	dryingSectionGroup3SteamPressureKp : REAL := 1.0;  // PID Kp for Group 1 steam pressure
	dryingSectionGroup3SteamPressureTn : REAL := 8.0;  // PID Tn for Group 1 steam pressure
	dryingSectionGroup3SteamPressureTv : REAL := 0.0;  // PID Tv for Group 1 steam pressure	

	
	dryingSectionGroup1TorqueKp : REAL := 1.0;  // PID Kp for Group 1 steam pressure
	dryingSectionGroup1TorqueTn : REAL := 8.0;  // PID Tn for Group 1 steam pressure
	dryingSectionGroup1TorqueTv : REAL := 0.0;  // PID Tv for Group 1 steam pressure
	
	dryingSectionGroup2TorqueKp : REAL := 1.0;  // PID Kp for Group 1 steam pressure
	dryingSectionGroup2TorqueTn : REAL := 8.0;  // PID Tn for Group 1 steam pressure
	dryingSectionGroup2TorqueTv : REAL := 0.0;  // PID Tv for Group 1 steam pressure
	
	dryingSectionGroup3TorqueKp : REAL := 1.0;  // PID Kp for Group 1 steam pressure
	dryingSectionGroup3TorqueTn : REAL := 8.0;  // PID Tn for Group 1 steam pressure
	dryingSectionGroup3TorqueTv : REAL := 0.0;  // PID Tv for Group 1 steam pressure
	
	
		
	firstPressDiameter	: REAL := 531.0;
	secondPressDiameter	: REAL := 800.9;	

	formingBoardSuctionRollDiameter		: REAL := 530.0;
	formingBoardTractionRollDiameter	: REAL := 580.0;
    tractionRollToSuctionRollGearRatio  : REAL := 0.915;

	formingBoardSuctionRollMotorRPM		: REAL := 329.3;
	formingBoardTractionRollMotorRPM	: REAL := 360.4;
	formingBoardTorqueDif				: REAL := 1.0;

	
	    //----------------------------------------------------------------------
    // PID GAINS
    //----------------------------------------------------------------------
    formingBoardTorquePIDCtrlKp                   : REAL := 2.0;
    formingBoardTorquePIDCtrlTn                   : REAL := 8.0;
    formingBoardTorquePIDCtrlTv                   : REAL := 0.0;
    formingBoardTorqueLimit                   : REAL := 100.0;
	
	
    pressTorquePIDCtrlKp                   : REAL := 2.0;
    pressTorquePIDCtrlTn                   : REAL := 8.0;
    pressTorquePIDCtrlTv                   : REAL := 0.0;	
    pressTorqueLimit                   	: REAL := 100.0;	
	
    dryingSectionGroup1TorquePIDCtrlKp		: REAL := 2.0;
    dryingSectionGroup1TorquePIDCtrlTn	: REAL := 8.0;
    dryingSectionGroup1TorquePIDCtrlTv	: REAL := 0.0;
    dryingSectionGroup1TorqueLimit	: REAL := 100.0;

		
    dryingSectionGroup2TorquePIDCtrlKp	: REAL := 2.0;
    dryingSectionGroup2TorquePIDCtrlTn	: REAL := 8.0;
    dryingSectionGroup2TorquePIDCtrlTv	: REAL := 0.0;
    dryingSectionGroup2TorqueLimit	: REAL := 100.0;
			
	dryingSectionGroup3TorquePIDCtrlKp	: REAL := 2.0;
    dryingSectionGroup3TorquePIDCtrlTn	: REAL := 8.0;
    dryingSectionGroup3TorquePIDCtrlTv	: REAL := 0.0;
    dryingSectionGroup3TorqueLimit	: REAL := 100.0;
		
	
	

	
	dryingSectionGroup1UpperMasterDiameter	: REAL := 263.878;
	dryingSectionGroup1UpperSlave1Diameter	: REAL := 1200.980;
	dryingSectionGroup1LowerMasterDiameter	: REAL := 263.241;
	dryingSectionGroup1LowerSlave1Diameter	: REAL := 263.241;
	dryingSectionGroup2UpperMasterDiameter	: REAL := 264.196;
	dryingSectionGroup2UpperSlave1Diameter	: REAL := 264.196;
	dryingSectionGroup2LowerMasterDiameter	: REAL := 264.196;
	dryingSectionGroup2LowerSlave1Diameter	: REAL := 264.196;	
	dryingSectionGroup3UpperMasterDiameter	: REAL := 264.196;
	dryingSectionGroup3UpperSlave1Diameter	: REAL := 263.878;
	dryingSectionGroup3LowerMasterDiameter	: REAL := 263.878;
	dryingSectionGroup3LowerSlave1Diameter	: REAL := 263.241;

	
	dryingSectionGroup1UpperAndLowerSpeedCalibration   : REAL := -0.06 ;  // Bias [%] between upper and lower
	dryingSectionGroup2UpperAndLowerSpeedCalibration   : REAL := -0.06 ;  // Bias [%] between upper and lower
	dryingSectionGroup3UpperAndLowerSpeedCalibration   : REAL := -0.06 ;  // Bias [%] between upper and lower
	
	
	dryingSectionGroup1SlaveToMasterRatio	: REAL := 1;
	dryingSectionGroup2SlaveToMasterRatio	: REAL := 1;
	dryingSectionGroup3SlaveToMasterRatio	: REAL := 1;

	dryingSectionGroup1SlaveTorqueDif	: REAL := 1;
	dryingSectionGroup2SlaveTorqueDif	: REAL := 1;
	dryingSectionGroup3SlaveTorqueDif	: REAL := 1;
	

	
	firstPressMotorRPM	: REAL := 374.5;
	secondPressMotorRPM	: REAL := 238.7;	
	
	dryingSectionGroup1UpperMasterMotorRPM	: REAL := 750;
	dryingSectionGroup1UpperSlave1MotorRPM	: REAL := 750;

	dryingSectionGroup1LowerMasterMotorRPM	: REAL := 750;
	dryingSectionGroup1LowerSlave1MotorRPM	: REAL := 750;


	dryingSectionGroup2UpperMasterMotorRPM	: REAL := 750;
	dryingSectionGroup2UpperSlave1MotorRPM	: REAL := 750;

	dryingSectionGroup2LowerMasterMotorRPM	: REAL := 750;
	dryingSectionGroup2LowerSlave1MotorRPM	: REAL := 750;

	
	dryingSectionGroup3UpperMasterMotorRPM	: REAL := 750;
	dryingSectionGroup3UpperSlave1MotorRPM	: REAL := 750;
	
	dryingSectionGroup3LowerMasterMotorRPM	: REAL := 750;
	dryingSectionGroup3LowerSlave1MotorRPM	: REAL := 750;
	
	

	winderDiameter	: REAL := 800.9;
	winderMotorRPM	: REAL := 212.5; //Motor RPM  / Rel. Mecanicia (1700 / 8)
	

	winderRiderRollMovPressure : REAL := 9.0;
	
	
	winderRiderRollStartPressure : REAL := 1.0;
	winderRiderRollAdvTime : TIME := T#2S;

	
			
	END_STRUCT
END_TYPE

// ---- Function Blocks/PaperMachine/DataTypes/PaperMachine_TypeHmiCommands.TcDUT
TYPE PaperMachine_TypeHmiCommands :
STRUCT

    // ─────────────── GENERAL MACHINE COMMANDS ───────────────
    machineReset : BOOL; // General machine reset (Reset geral da máquina)

	
    // ─────────────── FORMING BOARD ───────────────
    formingBoardStart          : BOOL;  // Start forming board (Ligar mesa formadora)
    formingBoardStop           : BOOL;  // Stop forming board (Parar mesa formadora)
    formingBoardFastStop           : BOOL;  // Stop forming board (Parar mesa formadora)

    formingBoardAutoMan           : BOOL;  // Auto mode select (Modo automático)
    formingBoardSetpointMan    : REAL;  // Manual speed/flow setpoint (Setpoint manual)
    formingBoardProductionSpeed: REAL;  // Select production (fast) speed (Selecionar velocidade de produção - rápida)
    formingBoardRollUpCmd      : BOOL;  // Command to raise/roll up forming board (Comando para subir mesa formadora)
    formingBoardRollDownCmd    : BOOL;  // Command to lower/roll down forming board (Comando para descer mesa formadora)

	// Automatic positioning (for auto mode)
	headboxLipsTargetSetpoint_mm       : REAL;          // Desired lips opening [mm]
	headboxLipsAutoAdjustCmd           : BOOL;          // Pulse to start auto adjustment
	// Manual jog commands (for manual mode)
	headboxLipsManualOpenCmd           : BOOL;          // Jog open while pressed
	headboxLipsManualCloseCmd          : BOOL;          // Jog close while pressed		
	
	formingTailCutterNozzleStartCmd   : BOOL; 
	formingTailCutterNozzleStopCmd   : BOOL; 
	
	formingTailCutterNozzleFwCmd   : BOOL; 
	formingTailCutterNozzleRevCmd   : BOOL; 	
	
	
	
	formingWireShowerStartCmd : BOOL; 
	formingWireShowerStopCmd : BOOL; 
	
	
	// ─────────────── PRESS SECTION ───────────────
	// Start/stop and speed control commands for the press section.
	pressSectionStart            : BOOL;  // Start Press Section (Ligar Prensa)
	pressSectionStop             : BOOL;  // Stop Press Section (Parar Prensa)
	pressSectionFastStop             : BOOL;  // Stop Press Section (Parar Prensa)

	pressSectionAutoMan          : BOOL;  // 1 = Auto / 0 = Manual mode (Modo automático/manual)
	pressSectionManualSetpoint   : REAL;  // Manual speed setpoint [m/min] (Setpoint manual)
	pressSectionSpeedInc         : BOOL;  // Increase speed manually (Aumentar velocidade)
	pressSectionSpeedDec         : BOOL;  // Decrease speed manually (Diminuir velocidade)
	pressSectionRecoverSpeedCmd  : BOOL;  // Temporarily recover speed (Recuperar velocidade)
	pressSectionRecoverIncrement : REAL;  // Recovery speed increment [m/min or %] (Incremento de recuperação)

	
	// ─────────────── DRYING SECTION — GROUP 1 ───────────────
	// Start/stop and speed control commands for the drying section (Group 1).
	dryingSectionGroup1Start            : BOOL;  // Start Drying Section Group 1 (Ligar Secagem Grupo 1)
	dryingSectionGroup1Stop             : BOOL;  // Stop Drying Section Group 1 (Parar Secagem Grupo 1)
	dryingSectionGroup1FastStop             : BOOL;  // Stop Drying Section Group 1 (Parar Secagem Grupo 1)

	dryingSectionGroup1AutoMan          : BOOL;  // 1 = Auto / 0 = Manual mode for Group 1 (Modo automático/manual Grupo 1)
	dryingSectionGroup1ManualSetpoint   : REAL;  // Manual speed setpoint [m/min] (Setpoint manual Grupo 1)
	dryingSectionGroup1SpeedInc         : BOOL;  // Increase Group 1 speed manually (Aumentar velocidade Grupo 1)
	dryingSectionGroup1SpeedDec         : BOOL;  // Decrease Group 1 speed manually (Diminuir velocidade Grupo 1)
	dryingSectionGroup1RecoverSpeedCmd  : BOOL;  // Temporarily recover speed (Recuperar velocidade Grupo 1)
	Group1RecoverIncrement : REAL;  // Recovery speed increment [m/min or %] (Incremento de recuperação Grupo 1)
	dryingSectionGroup1SteamPressureAutoMan : BOOL;  // Recovery speed increment [m/min or %] (Incremento de recuperação Grupo 1)
	dryingSectionGroup1SteamPressureAutoSetpoint : REAL;  // Recovery speed increment [m/min or %] (Incremento de recuperação Grupo 1)
	dryingSectionGroup1SteamPressureManualSetpoint : REAL;  // Recovery speed increment [m/min or %] (Incremento de recuperação Grupo 1)
	dryingSectionGroup1PaperBreakSteamPressure1 : REAL;  // Recovery speed increment [m/min or %] (Incremento de recuperação Grupo 1)
	dryingSectionGroup1PaperBreakSteamPressure2 : REAL;  // Recovery speed increment [m/min or %] (Incremento de recuperação Grupo 1)

	
	// ─────────────── DRYING SECTION — GROUP 2 ───────────────
	// Start/stop and speed control commands for the drying section (Group 2).
	dryingSectionGroup2Start            : BOOL;  // Start Drying Section Group 2 (Ligar Secagem Grupo 2)
	dryingSectionGroup2Stop             : BOOL;  // Stop Drying Section Group 2 (Parar Secagem Grupo 2)
	dryingSectionGroup2FastStop             : BOOL;  // Stop Drying Section Group 1 (Parar Secagem Grupo 1)

	dryingSectionGroup2AutoMan          : BOOL;  // 1 = Auto / 0 = Manual mode for Group 2 (Modo automático/manual Grupo 2)

	dryingSectionGroup2ManualSetpoint   : REAL;  // Manual speed setpoint [m/min] (Setpoint manual Grupo 2)
	dryingSectionGroup2SpeedInc         : BOOL;  // Increase Group 2 speed manually (Aumentar velocidade Grupo 2)
	dryingSectionGroup2SpeedDec         : BOOL;  // Decrease Group 2 speed manually (Diminuir velocidade Grupo 2)
	dryingSectionGroup2RecoverSpeedCmd  : BOOL;  // Temporarily recover speed (Recuperar velocidade Grupo 2)
	dryingSectionGroup2RecoverIncrement : REAL;  // Recovery speed increment [m/min or %] (Incremento de recuperação Grupo 2)
	dryingSectionGroup2SteamPressureAutoMan : BOOL;  // Recovery speed increment [m/min or %] (Incremento de recuperação Grupo 1)
	dryingSectionGroup2SteamPressureAutoSetpoint : REAL;  // Recovery speed increment [m/min or %] (Incremento de recuperação Grupo 1)
	dryingSectionGroup2SteamPressureManualSetpoint : REAL;  // Recovery speed increment [m/min or %] (Incremento de recuperação Grupo 1)
	dryingSectionGroup2PaperBreakSteamPressure1 : REAL;  // Recovery speed increment [m/min or %] (Incremento de recuperação Grupo 1)
	dryingSectionGroup2PaperBreakSteamPressure2 : REAL;  // Recovery speed increment [m/min or %] (Incremento de recuperação Grupo 1)
	
	// ─────────────── DRYING SECTION — GROUP 3 ───────────────
	// Start/stop and speed control commands for the drying section (Group 2).
	dryingSectionGroup3Start            : BOOL;  // Start Drying Section Group 2 (Ligar Secagem Grupo 2)
	dryingSectionGroup3Stop             : BOOL;  // Stop Drying Section Group 2 (Parar Secagem Grupo 2)
	dryingSectionGroup3FastStop             : BOOL;  // Stop Drying Section Group 1 (Parar Secagem Grupo 1)

	dryingSectionGroup3AutoMan          : BOOL;  // 1 = Auto / 0 = Manual mode for Group 2 (Modo automático/manual Grupo 2)
	dryingSectionGroup3ManualSetpoint   : REAL;  // Manual speed setpoint [m/min] (Setpoint manual Grupo 2)
	dryingSectionGroup3SpeedInc         : BOOL;  // Increase Group 2 speed manually (Aumentar velocidade Grupo 2)
	dryingSectionGroup3SpeedDec         : BOOL;  // Decrease Group 2 speed manually (Diminuir velocidade Grupo 2)
	dryingSectionGroup3RecoverSpeedCmd  : BOOL;  // Temporarily recover speed (Recuperar velocidade Grupo 2)
	dryingSectionGroup3RecoverIncrement : REAL;  // Recovery speed increment [m/min or %] (Incremento de recuperação Grupo 2)
	dryingSectionGroup3SteamPressureAutoMan : BOOL;  // Recovery speed increment [m/min or %] (Incremento de recuperação Grupo 1)
	dryingSectionGroup3SteamPressureAutoSetpoint : REAL;  // Recovery speed increment [m/min or %] (Incremento de recuperação Grupo 1)
	dryingSectionGroup3SteamPressureManualSetpoint : REAL;  // Recovery speed increment [m/min or %] (Incremento de recuperação Grupo 1)
	dryingSectionGroup3PaperBreakSteamPressure1 : REAL;  // Recovery speed increment [m/min or %] (Incremento de recuperação Grupo 1)
	dryingSectionGroup3PaperBreakSteamPressure2 : REAL;  // Recovery speed increment [m/min or %] (Incremento de recuperação Grupo 1)
	
    // ─────────────── DRYING SECTION - LUBRIFICATION UNIT ───────────────
    dryingSectionLubricationPumpStart      : BOOL;  // EN: Start command for lubrication unit (HMI → FB) / PT: Comando de PARTIDA da unidade de lubrificação (IHM → FB)
    dryingSectionLubricationPumpStop       : BOOL;  // EN: Stop command for lubrication unit (HMI → FB) / PT: Comando de PARADA da unidade de lubrificação (IHM → FB)
    dryingSectionLubricationPumpSelector   : BOOL;  // EN: Pump selector (FALSE = Pump 1, TRUE = Pump 2) / PT: Seletor de bomba (FALSE = Bomba 1, TRUE = Bomba 2)
    dryingSectionLubricationPumpAutoMan    : BOOL;  // EN: Mode selection (FALSE = Manual, TRUE = Automatic) / PT: Seleção de modo (FALSE = Manual, TRUE = Automático)

	// ─────────────── WINDER SECTION ───────────────
	// Start/stop and speed control commands for the winder section.
	winderSectionStart            : BOOL;  // Start Press Section (Ligar Prensa)
	winderSectionStop             : BOOL;  // Stop Press Section (Parar Prensa)
	winderSectionAutoMan          : BOOL;  // 1 = Auto / 0 = Manual mode (Modo automático/manual)
	winderSectionManualSetpoint   : REAL;  // Manual speed setpoint [m/min] (Setpoint manual)
	winderSectionSpeedInc         : BOOL;  // Increase speed manually (Aumentar velocidade)
	winderSectionSpeedDec         : BOOL;  // Decrease speed manually (Diminuir velocidade)
	winderSectionRecoverSpeedCmd  : BOOL;  // Temporarily recover speed (Recuperar velocidade)
	winderSectionRecoverIncrement : REAL;  // Recovery speed increment [m/min or %] (Incremento de recuperação)


	
	
	
  // Pressure fine adjustments for rider roll
    winderPressureOperatorSideIncCmd : BOOL; // EN: Increase operator-side pressure / PT: Aumenta a pressão no lado do operador
    winderPressureOperatorSideDecCmd : BOOL; // EN: Decrease operator-side pressure / PT: Diminui a pressão no lado do operador

    winderPressureDriveSideIncCmd    : BOOL; // EN: Increase drive-side pressure / PT: Aumenta a pressão no lado motriz
    winderPressureDriveSideDecCmd    : BOOL; // EN: Decrease drive-side pressure / PT: Diminui a pressão no lado motriz

	winderRiderRollWorkPositionCmd	: BOOL;
	winderRiderRollReleasePositionCmd	: BOOL;
	winderEnableTorqueControlCmd			: BOOL;

	winderTorqueSetpoint			: REAL;
	
    //==============================================================
    // CORE LOCK (CHUCK LOCKING SYSTEM)
    //==============================================================
    winderCoreLockAutoMan         : BOOL;  // EN: Core lock mode (0=Manual, 1=Auto) / PT: Modo do travamento do mandril (0=Manual, 1=Automático)
    winderCoreLockCmd             : BOOL;  // EN: Lock core chucks / PT: Travar mandril (core chucks)
    winderCoreUnlockCmd           : BOOL;  // EN: Unlock core chucks / PT: Destravar mandril

	//==============================================================
    // CORE LOCK (CHUCK LOCKING SYSTEM)
    //==============================================================
	winderCoreAceleratorEngageCmd : BOOL;
	winderCoreAceleratorDisengageCmd : BOOL;
	
    //==============================================================
    // CORE BRAKE CONTROL
    //==============================================================
    winderCoreBrakeAutoMan        : BOOL;  // EN: Core brake mode (0=Manual, 1=Auto) / PT: Modo de freio do mandril (0=Manual, 1=Automático)
    winderCoreBrakeEnableCmd      : BOOL;  // EN: Enable core brake / PT: Habilita o freio do mandril
    winderCoreBrakeDisableCmd     : BOOL;  // EN: Disable core brake / PT: Desabilita o freio do mandril	
	
	winderCorePositioningArmFwdCmd      : BOOL;  // EN: Command to move arm forward / PT: Comando para avançar o braço posicionador
    winderCorePositioningArmRevCmd      : BOOL;  // EN: Command to move arm backward / PT: Comando para recuar o braço posicionador

    winderCorePositioningArmPosLimitFwd : BOOL;  // EN: Forward limit switch / PT: Fim de curso avançado
    winderCorePositioningArmPosLimitRev : BOOL;  // EN: Reverse limit switch / PT: Fim de curso recuado
	
    // ─────────────── CENTRIFUGAL PRESSURE SCREEN ───────────────
    pressureScreenStart : BOOL;  // Start centrifugal pressure screen (Ligar peneira centrífuga de pressão)
    pressureScreenStop  : BOOL;  // Stop centrifugal pressure screen (Parar peneira centrífuga de pressão)
	

    // ─────────────── COUCH PIT PUMP & MIXER ───────────────
    couchPitPumpStart        : BOOL;  // Start couch pit pump (Ligar bomba do poço da mesa couch)
    couchPitPumpStop         : BOOL;  // Stop couch pit pump (Parar bomba do poço da mesa couch)
    couchPitPumpAutoMan      : BOOL;  // Auto/manual mode select (Seleção automático/manual)
    couchPitPumpSetpointMan  : REAL;  // Manual setpoint (Setpoint manual)
    couchPitPumpSetpointAuto : REAL;  // Auto setpoint (Setpoint automático)
    couchPitMixerStart       : BOOL;  // Start couch pit mixer (Ligar misturador do poço da mesa couch)
    couchPitMixerStop        : BOOL;  // Stop couch pit mixer (Parar misturador do poço da mesa couch)

    // ─────────────── WIRE PIT PUMP ───────────────
    wirePitPumpStart    : BOOL;  // Start wire pit pump (Ligar bomba do poço da mesa plana)
    wirePitPumpStop     : BOOL;  // Stop wire pit pump (Parar bomba do poço da mesa plana)
    wirePitPumpAutoMan  : BOOL;  // Auto/manual mode select (Seleção automático/manual)
    wirePitSetpointMan  : REAL;  // Manual setpoint (Setpoint manual)
    wirePitSetpointManInc  : BOOL;  // Manual setpoint (Setpoint manual)
    wirePitSetpointManDec  : BOOL;  // Manual setpoint (Setpoint manual)	
    wirePitSetpointAuto 	: REAL;  // Auto setpoint (Setpoint automático)
    wirePitSetpointAutoInc  : BOOL;  // Manual setpoint (Setpoint manual)
    wirePitSetpointAutoDec  : BOOL;  // Manual setpoint (Setpoint manual)	

	
	whiteWaterSiloAutoMan           : BOOL;  // Auto/manual mode select (Seleção automático/manual)
	
	// --- Manual setpoint (e.g., level %, flow m3/h, or pressure) ---
	whiteWaterSiloSetpointMan       : REAL;  // Manual setpoint (Setpoint manual)
	whiteWaterSiloSetpointManInc    : BOOL;  // Manual setpoint increase command (Incrementar setpoint manual)
	whiteWaterSiloSetpointManDec    : BOOL;  // Manual setpoint decrease command (Decrementar setpoint manual)
	
	// --- Auto setpoint (from recipe / process / cascade control) ---
	whiteWaterSiloSetpointAuto      : REAL;  // Auto setpoint (Setpoint automático)
	whiteWaterSiloSetpointAutoInc   : BOOL;  // Auto setpoint increase command (Incrementar setpoint automático)
	whiteWaterSiloSetpointAutoDec   : BOOL;  // Auto setpoint decrease command (Decrementar setpoint automático)	
	
	
    // ─────────────── STOCK PUMP ───────────────
    stockPumpStart        : BOOL;  // Start stock pump (Ligar bomba de massa)
    stockPumpStop         : BOOL;  // Stop stock pump (Parar bomba de massa)
    stockPumpAutoMan      : BOOL;  // Auto/manual mode select (Seleção automático/manual)
    stockPumpSetpointMan  : REAL;  // Manual setpoint (Setpoint manual)
    stockPumpSetpointManInc  : BOOL;  // Manual setpoint (Setpoint manual)
    stockPumpSetpointManDec  : BOOL;  // Manual setpoint (Setpoint manual)
	
    stockPumpSetpointAuto : REAL;  // Auto setpoint (Setpoint automático)
    stockPumpSetpointAutoInc : BOOL;  // Auto setpoint (Setpoint automático)
    stockPumpSetpointAutoDec : BOOL;  // Auto setpoint (Setpoint automático)
	

    // ─────────────── MIX PUMP ───────────────
    mixPumpStart      : BOOL;  // Start mixing pump (Ligar bomba de mistura)
    mixPumpStop       : BOOL;  // Stop mixing pump (Parar bomba de mistura)
    mixPumpAutoMan    : BOOL;  // Auto/manual mode select (Seleção automático/manual)
	mixPumpSetpointManInc: BOOL;  // Manual setpoint (Setpoint manual)
	mixPumpSetpointManDec: BOOL;  // Manual setpoint (Setpoint manual)
	mixPumpRatioInc   : BOOL;  // Increase mix ratio (Aumentar proporção de mistura)
    mixPumpRatioDec   : BOOL;  // Decrease mix ratio (Diminuir proporção de mistura)
	mixPumpSetpointMan: REAL;  // Manual setpoint (Setpoint manual)
	mixPumpRatio   	: REAL;  // Increase mix ratio (Aumentar proporção de mistura)

    // ─────────────── VACUUM PUMPS ───────────────
    vacuumSealPumpStart      : BOOL;  // Start vacuum seal pump (Ligar bomba de vedação a vácuo)
    vacuumSealPumpStop       : BOOL;  // Stop vacuum seal pump (Parar bomba de vedação a vácuo)
    vacuumWaterSepPumpStart  : BOOL;  // Start water separator vacuum pump (Ligar bomba de vácuo separadora de água)
    vacuumWaterSepPumpStop   : BOOL;  // Stop water separator vacuum pump (Parar bomba de vácuo separadora de água)
    suctionRollVacuumPumpStart: BOOL; // Start suction roll vacuum pump (Ligar bomba de vácuo do rolo de sucção)
    suctionRollVacuumPumpStop : BOOL; // Stop suction roll vacuum pump (Parar bomba de vácuo do rolo de sucção)
    wireVacuumPumpStart      : BOOL;  // Start wire section vacuum pump (Ligar bomba de vácuo da mesa plana)
    wireVacuumPumpStop       : BOOL;  // Stop wire section vacuum pump (Parar bomba de vácuo da mesa plana)
    pressVacuumPump1Start     : BOOL;  // Start press section vacuum pump (Ligar bomba de vácuo da seção de prensas)
    pressVacuumPump1Stop      : BOOL;  // Stop press section vacuum pump (Parar bomba de vácuo da seção de prensas)
    pressVacuumPump2Start     : BOOL;  // Start press section vacuum pump (Ligar bomba de vácuo da seção de prensas)
    pressVacuumPump2Stop      : BOOL;  // Stop press section vacuum pump (Parar bomba de vácuo da seção de prensas)

    // ─────────────── LOW VACUUM EXHAUST FAN ───────────────
    lowVacuumExhaustFanStart : BOOL;  // Start low vacuum exhaust fan (Ligar exaustor do baixo vácuo)
    lowVacuumExhaustFanStop  : BOOL;  // Stop low vacuum exhaust fan (Parar exaustor do baixo vácuo)

    // ─────────────── WIRE SECTION ───────────────
    wireSectionDisplacementOpSide    : BOOL;  // Displacement sensor - operator side (Sensor de deslocamento - lado operador)
    wireSectionDisplacementDriveSide : BOOL;  // Displacement sensor - drive side (Sensor de deslocamento - lado acionamento)
    wireSectionTensionLimitMax       : REAL;  // Maximum wire tension limit (Limite máximo de tensão da tela formadora)
    wireSectionTensionLimitMin       : REAL;  // Minimum wire tension limit (Limite mínimo de tensão da tela formadora)
    wireSectionStretchExtendCmd      : BOOL;  // Command to stretch wire (Comando para esticar a tela)
    wireSectionStretchReleaseCmd     : BOOL;  // Command to release wire (Comando para aliviar a tela)

END_STRUCT
END_TYPE

// ---- Function Blocks/PaperMachine/DataTypes/PaperMachine_TypeHmiStatus.TcDUT
TYPE PaperMachine_TypeHmiStatus :
STRUCT

	alarmIndication	: BOOL; //Used to tell the hmi that we have an alarm active

    // ─────────────── FORMING LIPS OPENNING CONTROL ───────────────
	headboxLipsPosition_mm       		  : REAL;  // Head box lips position [mm]
	
    // ─────────────── FORMING BOARD ROLLS ───────────────
    formingBoardSuctionRollSpeed    : REAL;  // Suction roll speed (Velocidade do rolo de sucção)
    formingBoardSuctionRollTorque   : REAL;  // Suction roll torque (Torque do rolo de sucção)
    formingBoardSuctionRollState   	: INT;  // Suction roll state 

    formingBoardTractionRollSpeed   : REAL;  // Traction roll speed (Velocidade do rolo tracionador)
    formingBoardTractionRollTorque  : REAL;  // Traction roll torque (Torque do rolo tracionador)
    formingBoardTractionRollState  	: INT;  // Traction roll state 
	
	formingTailCutterNozzleState   : INT; 
	formingWireShowerState : INT; 
	
	// ─────────────── PRESS SECTION DRIVES ───────────────
	firstPressSectionSpeed     : REAL;  // First Press (Master) speed [m/min or rpm] (Velocidade do rolo prensador 1 - mestre)
	firstPressSectionTorque    : REAL;  // First Press (Master) torque [% or Nm] (Torque do rolo prensador 1 - mestre)
	firstPressSectionState     : INT;   // First Press (Master) state code (Estado do rolo prensador 1 - mestre)
	
	secondPressSectionSpeed    : REAL;  // Second Press (Slave) speed [m/min or rpm] (Velocidade do rolo prensador 2 - escravo)
	secondPressSectionTorque   : REAL;  // Second Press (Slave) torque [% or Nm] (Torque do rolo prensador 2 - escravo)
	secondPressSectionState    : INT;   // Second Press (Slave) state code (Estado do rolo prensador 2 - escravo)
	presseGroupSpeedDif				: REAL;	
		
	
	// ─────────────── DRYING SECTION — GROUP 1 ───────────────
	// Speed, torque, and state variables for upper and lower groups of Drying Section Group 1.
	
	// ── UPPER GROUP (GROUP 1) ────────────────────────────────────────────────
	dryingSectionGroup1UpperMasterSpeedMPM   : REAL;  // Group 1 Upper Master speed [m/min or rpm] (Velocidade do motor mestre superior do grupo 1)
	dryingSectionGroup1UpperMasterTorque  : REAL;  // Group 1 Upper Master torque [% or Nm] (Torque do motor mestre superior do grupo 1)
	dryingSectionGroup1UpperMasterState   : INT;   // Group 1 Upper Master state code (Estado do motor mestre superior do grupo 1)
	
	dryingSectionGroup1UpperSlave1SpeedMPM   : REAL;  // Group 1 Upper Slave 1 speed [m/min or rpm] (Velocidade do motor escravo 1 superior do grupo 1)
	dryingSectionGroup1UpperSlave1Torque  : REAL;  // Group 1 Upper Slave 1 torque [% or Nm] (Torque do motor escravo 1 superior do grupo 1)
	dryingSectionGroup1UpperSlave1State   : INT;   // Group 1 Upper Slave 1 state code (Estado do motor escravo 1 superior do grupo 1)
	
	dryingSectionGroup1UpperSlave2SpeedMPM   : REAL;  // Group 1 Upper Slave 2 speed [m/min or rpm] (Velocidade do motor escravo 2 superior do grupo 1)
	dryingSectionGroup1UpperSlave2Torque  : REAL;  // Group 1 Upper Slave 2 torque [% or Nm] (Torque do motor escravo 2 superior do grupo 1)
	dryingSectionGroup1UpperSlave2State   : INT;   // Group 1 Upper Slave 2 state code (Estado do motor escravo 2 superior do grupo 1)
	
	
	// ── LOWER GROUP (GROUP 1) ────────────────────────────────────────────────
	dryingSectionGroup1LowerMasterSpeedMPM   : REAL;  // Group 1 Lower Master speed [m/min or rpm] (Velocidade do motor mestre inferior do grupo 1)
	dryingSectionGroup1LowerMasterTorque  : REAL;  // Group 1 Lower Master torque [% or Nm] (Torque do motor mestre inferior do grupo 1)
	dryingSectionGroup1LowerMasterState   : INT;   // Group 1 Lower Master state code (Estado do motor mestre inferior do grupo 1)
	
	dryingSectionGroup1LowerSlave1SpeedMPM   : REAL;  // Group 1 Lower Slave 1 speed [m/min or rpm] (Velocidade do motor escravo 1 inferior do grupo 1)
	dryingSectionGroup1LowerSlave1Torque  : REAL;  // Group 1 Lower Slave 1 torque [% or Nm] (Torque do motor escravo 1 inferior do grupo 1)
	dryingSectionGroup1LowerSlave1State   : INT;   // Group 1 Lower Slave 1 state code (Estado do motor escravo 1 inferior do grupo 1)
	
	dryingSectionGroup1LowerSlave2SpeedMPM   : REAL;  // Group 1 Lower Slave 2 speed [m/min or rpm] (Velocidade do motor escravo 2 inferior do grupo 1)
	dryingSectionGroup1LowerSlave2Torque  : REAL;  // Group 1 Lower Slave 2 torque [% or Nm] (Torque do motor escravo 2 inferior do grupo 1)
	dryingSectionGroup1LowerSlave2State   : INT;   // Group 1 Lower Slave 2 state code (Estado do motor escravo 2 inferior do grupo 1)
	
	dryingSectionGroup1SteamPressure   : REAL;   // Drying group 1 - Steam pressure display
	dryingSectionGroup1SpeedDif				: REAL;	

	dryingSectionGroup1PaperPresence				: BOOL;	
	
	
	// ─────────────── DRYING SECTION — GROUP 2 ───────────────
	// Speed, torque, and state variables for upper and lower groups of Drying Section Group 2.
	
	// ── UPPER GROUP (GROUP 2) ────────────────────────────────────────────────
	dryingSectionGroup2UpperMasterSpeedMPM   : REAL;  // Group 2 Upper Master speed [m/min or rpm] (Velocidade do motor mestre superior do grupo 2)
	dryingSectionGroup2UpperMasterTorque  : REAL;  // Group 2 Upper Master torque [% or Nm] (Torque do motor mestre superior do grupo 2)
	dryingSectionGroup2UpperMasterState   : INT;   // Group 2 Upper Master state code (Estado do motor mestre superior do grupo 2)
	
	dryingSectionGroup2UpperSlave1SpeedMPM   : REAL;  // Group 2 Upper Slave 1 speed [m/min or rpm] (Velocidade do motor escravo 1 superior do grupo 2)
	dryingSectionGroup2UpperSlave1Torque  : REAL;  // Group 2 Upper Slave 1 torque [% or Nm] (Torque do motor escravo 1 superior do grupo 2)
	dryingSectionGroup2UpperSlave1State   : INT;   // Group 2 Upper Slave 1 state code (Estado do motor escravo 1 superior do grupo 2)
	
	dryingSectionGroup2UpperSlave2Speed   : REAL;  // Group 2 Upper Slave 2 speed [m/min or rpm] (Velocidade do motor escravo 2 superior do grupo 2)
	dryingSectionGroup2UpperSlave2Torque  : REAL;  // Group 2 Upper Slave 2 torque [% or Nm] (Torque do motor escravo 2 superior do grupo 2)
	dryingSectionGroup2UpperSlave2State   : INT;   // Group 2 Upper Slave 2 state code (Estado do motor escravo 2 superior do grupo 2)
	
	
	// ── LOWER GROUP (GROUP 2) ────────────────────────────────────────────────
	dryingSectionGroup2LowerMasterSpeedMPM   : REAL;  // Group 2 Lower Master speed [m/min or rpm] (Velocidade do motor mestre inferior do grupo 2)
	dryingSectionGroup2LowerMasterTorque  : REAL;  // Group 2 Lower Master torque [% or Nm] (Torque do motor mestre inferior do grupo 2)
	dryingSectionGroup2LowerMasterState   : INT;   // Group 2 Lower Master state code (Estado do motor mestre inferior do grupo 2)
	
	dryingSectionGroup2LowerSlave1SpeedMPM   : REAL;  // Group 2 Lower Slave 1 speed [m/min or rpm] (Velocidade do motor escravo 1 inferior do grupo 2)
	dryingSectionGroup2LowerSlave1Torque  : REAL;  // Group 2 Lower Slave 1 torque [% or Nm] (Torque do motor escravo 1 inferior do grupo 2)
	dryingSectionGroup2LowerSlave1State   : INT;   // Group 2 Lower Slave 1 state code (Estado do motor escravo 1 inferior do grupo 2)
	
	dryingSectionGroup2LowerSlave2SpeedMPM   : REAL;  // Group 2 Lower Slave 2 speed [m/min or rpm] (Velocidade do motor escravo 2 inferior do grupo 2)
	dryingSectionGroup2LowerSlave2Torque  : REAL;  // Group 2 Lower Slave 2 torque [% or Nm] (Torque do motor escravo 2 inferior do grupo 2)
	dryingSectionGroup2LowerSlave2State   : INT;   // Group 2 Lower Slave 2 state code (Estado do motor escravo 2 inferior do grupo 2)
	
	dryingSectionGroup2SteamPressure   : REAL;   // Drying group 1 - Steam pressure display
	dryingSectionGroup2SpeedDif				: REAL;	
		
	dryingSectionGroup2PaperPresence				: BOOL;	
	
	// ─────────────── DRYING SECTION — GROUP 3 ───────────────
	// Speed, torque, and state variables for upper and lower groups of Drying Section Group 2.
	
	// ── UPPER GROUP (GROUP 3) ────────────────────────────────────────────────
	dryingSectionGroup3UpperMasterSpeedMPM   : REAL;  // Group 2 Upper Master speed [m/min or rpm] (Velocidade do motor mestre superior do grupo 2)
	dryingSectionGroup3UpperMasterTorque  : REAL;  // Group 2 Upper Master torque [% or Nm] (Torque do motor mestre superior do grupo 2)
	dryingSectionGroup3UpperMasterState   : INT;   // Group 2 Upper Master state code (Estado do motor mestre superior do grupo 2)
	
	dryingSectionGroup3UpperSlave1SpeedMPM   : REAL;  // Group 2 Upper Slave 1 speed [m/min or rpm] (Velocidade do motor escravo 1 superior do grupo 2)
	dryingSectionGroup3UpperSlave1Torque  : REAL;  // Group 2 Upper Slave 1 torque [% or Nm] (Torque do motor escravo 1 superior do grupo 2)
	dryingSectionGroup3UpperSlave1State   : INT;   // Group 2 Upper Slave 1 state code (Estado do motor escravo 1 superior do grupo 2)
	
	dryingSectionGroup3UpperSlave2SpeedMPM   : REAL;  // Group 2 Upper Slave 2 speed [m/min or rpm] (Velocidade do motor escravo 2 superior do grupo 2)
	dryingSectionGroup3UpperSlave2Torque  : REAL;  // Group 2 Upper Slave 2 torque [% or Nm] (Torque do motor escravo 2 superior do grupo 2)
	dryingSectionGroup3UpperSlave2State   : INT;   // Group 2 Upper Slave 2 state code (Estado do motor escravo 2 superior do grupo 2)
	
	
	// ── LOWER GROUP (GROUP 3) ────────────────────────────────────────────────
	dryingSectionGroup3LowerMasterSpeedMPM   : REAL;  // Group 2 Lower Master speed [m/min or rpm] (Velocidade do motor mestre inferior do grupo 2)
	dryingSectionGroup3LowerMasterTorque  : REAL;  // Group 2 Lower Master torque [% or Nm] (Torque do motor mestre inferior do grupo 2)
	dryingSectionGroup3LowerMasterState   : INT;   // Group 2 Lower Master state code (Estado do motor mestre inferior do grupo 2)
	
	dryingSectionGroup3LowerSlave1SpeedMPM   : REAL;  // Group 2 Lower Slave 1 speed [m/min or rpm] (Velocidade do motor escravo 1 inferior do grupo 2)
	dryingSectionGroup3LowerSlave1Torque  : REAL;  // Group 2 Lower Slave 1 torque [% or Nm] (Torque do motor escravo 1 inferior do grupo 2)
	dryingSectionGroup3LowerSlave1State   : INT;   // Group 2 Lower Slave 1 state code (Estado do motor escravo 1 inferior do grupo 2)
	
	dryingSectionGroup3LowerSlave2SpeedMPM   : REAL;  // Group 2 Lower Slave 2 speed [m/min or rpm] (Velocidade do motor escravo 2 inferior do grupo 2)
	dryingSectionGroup3LowerSlave2Torque  : REAL;  // Group 2 Lower Slave 2 torque [% or Nm] (Torque do motor escravo 2 inferior do grupo 2)
	dryingSectionGroup3LowerSlave2State   : INT;   // Group 2 Lower Slave 2 state code (Estado do motor escravo 2 inferior do grupo 2)

	dryingSectionGroup3SteamPressure   : REAL;   // Drying group 1 - Steam pressure display
	dryingSectionGroup3SpeedDif				: REAL;	
	dryingSectionGroup3PaperPresence				: BOOL;	
	
	
	winderPaperPresence				: BOOL;	

			
    // ─────────────── LUBRIFICATION UNIT ───────────────
    dryingSectionLubricationPump1State             : INT;   // EN: Pump 1 state (0=Stopped,1=Running,3=Fault) / PT: Estado da bomba 1 (0=Parada,1=Rodando,3=Falha)
    dryingSectionLubricationPump2State             : INT;   // EN: Pump 2 state (0=Stopped,1=Running,3=Fault) / PT: Estado da bomba 2 (0=Parada,1=Rodando,3=Falha)
    dryingSectionLubricationTankTemperature        : REAL;  // EN: Oil tank temperature [°C] / PT: Temperatura do tanque de óleo [°C]
    dryingSectionLubricationCircuitTemperature        : REAL;  // EN: Oil tank temperature [°C] / PT: Temperatura do tanque de óleo [°C]	
 
   // ─────────────── CENTRIFUGAL PRESSURE SCREEN ───────────────
    pressureScreenState             : INT;   // Centrifugal pressure screen state (Estado da peneira centrífuga de pressão)


    // ─────────────── COUCH PIT PUMP & MIXER ───────────────
    couchPitPumpState               : INT;   // Couch pit pump state (Estado da bomba do poço da mesa couch)
    couchPitPumpSpeed               : REAL;  // Couch pit pump speed (Velocidade da bomba do poço da mesa couch)
    couchPitPumpTorque              : REAL;  // Couch pit pump torque (Torque da bomba do poço da mesa couch)

    couchPitMixerState              : INT;   // Couch pit mixer state (Estado do agitador do poço da mesa couch)
    couchPitLevel             : REAL;  // Couch pit pump torque (Torque da bomba do poço da mesa couch)


    // ─────────────── WIRE PIT PUMP ───────────────
    wirePitPumpState                : INT;   // Wire pit pump state (Estado da bomba do poço da mesa plana)
    wirePitPumpSpeed                : REAL;  // Wire pit pump speed (Velocidade da bomba do poço da mesa plana)
    wirePitPumpTorque               : REAL;  // Wire pit pump torque (Torque da bomba do poço da mesa plana)
   	wirePitLevel             		: REAL;  // Couch pit pump torque (Torque da bomba do poço da mesa couch)

	
	// --- Manual setpoint (e.g., level %, flow m3/h, or pressure) ---
	whiteWaterSiloLevel       : REAL;  // Manual setpoint (Setpoint manual)
	whiteWaterSiloCtrlOutput       : REAL;  // Manual setpoint (Setpoint manual)

	

    // ─────────────── STOCK PUMP ───────────────
    stockPumpState                  : INT;   // Stock pump state (Estado da bomba de massa)
    stockPumpSpeed               	: REAL;  // Stock pump speed (Velocidade da bomba de massa)
    stockPumpTorque              	: REAL;  // Stock pump torque (Torque da bomba de massa)


    // ─────────────── MIXING PUMP ───────────────
    mixPumpState                    : INT;   // Mixing pump state (Estado da bomba de mistura)
    mixPumpSpeed                    : REAL;  // Mixing pump speed (Velocidade da bomba de mistura)
    mixPumpTorque                   : REAL;  // Mixing pump torque (Torque da bomba de mistura)
 	mixPumpSetpointMan				: REAL;  // Manual setpoint (Setpoint manual)

    // ─────────────── HEAD BOX ───────────────
	
    headBoxMMH2O                    : REAL;  // Pressure in mmH₂O (Pressão em mmH₂O)
    headBoxMMH2OCalc                : REAL;  // Calculated pressure in mmH₂O (Pressão calculada em mmH₂O)
    headBoxJetSpeedMPS                : REAL;  // Calculated pressure in mmH₂O (Pressão calculada em mmH₂O)
	
    mixPumpRatio                    : REAL;  // Mixing ratio (Relação de jato tela)
	
	

    // ─────────────── VACUUM PUMPS ───────────────
    vacuumSealPumpState             : INT;   // Vacuum seal pump state (Estado da bomba de vedação a vácuo)
    vacuumWaterSepPumpState         : INT;   // Water separator vacuum pump state (Estado da bomba de vácuo separadora de água)
    suctionRollVacuumPumpState      : INT;   // Suction roll vacuum pump state (Estado da bomba de vácuo do rolo de sucção)
    wireVacuumPumpState             : INT;   // Wire section vacuum pump state (Estado da bomba de vácuo da mesa plana)


	pressFeltVaccum1State			: INT;
	pressFeltVaccum2State			: INT;
	
	
    // ─────────────── LOW VACUUM EXHAUST FAN ───────────────
    lowVacuumExhaustFanState        : INT;   // Low vacuum exhaust fan state (Estado do exaustor de baixo vácuo)
	
	
	
	winderPressureSetpointOperatorSide : REAL; // EN: Controller output (operator side) / PT: Saída do controlador (lado operador)
    winderPressureSetpointDriveSide    : REAL; // EN: Controller output (drive side) / PT: Saída do controlador (lado motriz)
	winderSpeedMPM   : REAL;  // Group 2 Upper Slave 2 speed [m/min or rpm] (Velocidade do motor escravo 2 superior do grupo 2)
	winderTorque  : REAL;  // Group 2 Upper Slave 2 torque [% or Nm] (Torque do motor escravo 2 superior do grupo 2)
	winderState   : INT;   // Group 2 Upper Slave 2 state code (Estado do motor escravo 2 superior do grupo 2)
	winderSpeedDif				: REAL;	
		

	
	
END_STRUCT
END_TYPE

// ---- Function Blocks/PaperMachine/DataTypes/PaperMachine_TypeHmiAlarms.TcDUT
TYPE PaperMachine_TypeHmiAlarms :
STRUCT

	alarmIndication	: BOOL; //Used to tell the hmi that we have an alarm active

	
	formingBoardSafetyAlarm			: BOOL;
	pressSectionSafetyAlarm			: BOOL;
	dryingSectionSafetyAlarm		: BOOL;
	winderSectionSafetyAlarm		: BOOL;
	
    // ─────────────── FORMING BOARD ROLLS ───────────────
    formingBoardSuctionRollFaultAlarm         : BOOL;  // Suction roll fault / trip
    formingBoardSuctionRollCoolingFaultAlarm  : BOOL;  // Suction roll forced cooling fault
    formingBoardTractionRollFaultAlarm        : BOOL;  // Traction roll fault / trip
    formingBoardTractionRollCoolingFaultAlarm : BOOL;  // Traction roll forced cooling fault

    formingBoardRollDriveFaultAlarm           : BOOL;  // Roll up/down motor fault
    formingBoardStretchDriveFaultAlarm        : BOOL;  // Stretch motor fault
	formingBoardSpeedDifAlarm	: BOOL;

    // ── WIRE EDGE / RUNNING SAFETY SENSORS ─────────────────────────────────────
    formingBoardWireOverrunOperatorSideAlarm  : BOOL;  // Wire overrun detected on operator side (sensor active)
    formingBoardWireOverrunDriveSideAlarm     : BOOL;  // Wire overrun detected on drive side (sensor active)

    // ─────────────── PRESS SECTION DRIVES ───────────────
    pressSectionFirstPressFaultAlarm          : BOOL;  // First press (master) fault / trip
    pressSectionFirstPressCoolingFaultAlarm   : BOOL;  // First press forced cooling fault
    pressSectionSecondPressFaultAlarm         : BOOL;  // Second press (slave) fault / trip
    pressSectionSecondPressCoolingFaultAlarm  : BOOL;  // Second press forced cooling fault

    // ─────────────── PRESS SECTION — AUXILIARY MOTORS ───────────────
    pressSectionUpperFeltStretcherFaultAlarm  : BOOL;  // Upper felt stretcher motor fault / trip
    pressSectionLowerFeltStretcherFaultAlarm  : BOOL;  // Lower felt stretcher motor fault / trip
    pressSectionUpperInfeedRollFaultAlarm     : BOOL;  // Upper infeed roll motor fault / trip
    pressSectionLowerInfeedRollFaultAlarm     : BOOL;  // Lower infeed roll motor fault / trip

    // ── FELT EDGE / RUNNING SAFETY SENSORS ─────────────────────────────────────
    pressSectionUpperFelt1OverrunOperatorSideAlarm : BOOL;  // Felt 1 overrun detected on operator side (sensor active)
    pressSectionUpperFelt1OverrunDriveSideAlarm    : BOOL;  // Felt 1 overrun detected on drive side (sensor active)
    pressSectionUpperFelt2OverrunOperatorSideAlarm : BOOL;  // Felt 2 overrun detected on operator side (sensor active)
    pressSectionUpperFelt2OverrunDriveSideAlarm    : BOOL;  // Felt 2 overrun detected on drive side (sensor active)
    pressSectionLowerFeltOverrunOperatorSideAlarm  : BOOL;  // Felt 3 overrun detected on operator side (sensor active)
    pressSectionLowerFeltOverrunDriveSideAlarm     : BOOL;  // Felt 3 overrun detected on drive side (sensor active)

    // ─────────────── PRESS SECTION — GROUP FAULT ───────────────
    pressSectionGroupFaultAlarm               : BOOL;  // Global press section group fault / interlock active

    // ─────────────── DRYING SECTION — GROUP 1 ───────────────
    dryingSectionGroup1UpperMasterFaultAlarm         : BOOL;  // G1 Upper Master fault / trip
    dryingSectionGroup1UpperMasterCoolingFaultAlarm  : BOOL;  // G1 Upper Master forced cooling fault
    dryingSectionGroup1UpperSlave1FaultAlarm         : BOOL;  // G1 Upper Slave1 fault / trip
    dryingSectionGroup1UpperSlave1CoolingFaultAlarm  : BOOL;  // G1 Upper Slave1 forced cooling fault
    dryingSectionGroup1UpperSlave2FaultAlarm         : BOOL;  // G1 Upper Slave2 fault / trip
    dryingSectionGroup1UpperSlave2CoolingFaultAlarm  : BOOL;  // G1 Upper Slave2 forced cooling fault

    dryingSectionGroup1LowerMasterFaultAlarm         : BOOL;  // G1 Lower Master fault / trip
    dryingSectionGroup1LowerMasterCoolingFaultAlarm  : BOOL;  // G1 Lower Master forced cooling fault
    dryingSectionGroup1LowerSlave1FaultAlarm         : BOOL;  // G1 Lower Slave1 fault / trip
    dryingSectionGroup1LowerSlave1CoolingFaultAlarm  : BOOL;  // G1 Lower Slave1 forced cooling fault
    dryingSectionGroup1LowerSlave2FaultAlarm         : BOOL;  // G1 Lower Slave2 fault / trip
    dryingSectionGroup1LowerSlave2CoolingFaultAlarm  : BOOL;  // G1 Lower Slave2 forced cooling fault

    // ── FABRIC OVERRUN PROTECTION — GROUP 1 ───────────────────────────────────
    upperDryingSectionGroup1FabricOverrunOperatorSideAlarm : BOOL;  // Fabric overrun detected on operator side (sensor active)
    upperDryingSectionGroup1FabricOverrunDriveSideAlarm    : BOOL;  // Fabric overrun detected on drive side (sensor active)
    lowerDryingSectionGroup1FabricOverrunOperatorSideAlarm : BOOL;  // Fabric overrun detected on operator side (sensor active)
    lowerDryingSectionGroup1FabricOverrunDriveSideAlarm    : BOOL;  // Fabric overrun detected on drive side (sensor active)

    // ───────── DRYING SECTION — FABRIC STRETCHER — GROUP 1 ─────────
    upperDryingSectionGroup1FabricStretcherMotorFaultAlarm : BOOL;  // Upper fabric stretcher motor fault (G1)
    lowerDryingSectionGroup1FabricStretcherMotorFaultAlarm : BOOL;  // Lower fabric stretcher motor fault (G1)

    // ───────── DRYING SECTION — AUXILIARIES — GROUP 1 ─────────
    dryingSectionGroup1PickUpRollPosFaultAlarm       : BOOL;  // EN: G1 pick-up roll positioner fault / PT: Falha do posicionador do rolo pick-up G1
    dryingSectionGroup1BabyDryerScraperOscFaultAlarm : BOOL;  // EN: G1 babydryer scraper oscillator fault / PT: Falha do oscilador da raspa do babydryer G1
    dryingSectionGroup1UpperScraperOscFaultAlarm     : BOOL;  // EN: G1 upper group scraper oscillator fault / PT: Falha do oscilador da raspa do grupo superior G1
    dryingSectionGroup1LowerScraperOscFaultAlarm     : BOOL;  // EN: G1 lower group scraper oscillator fault / PT: Falha do oscilador da raspa do grupo inferior G1
	dryingSectionGroup1PaperBreakAlarm : BOOL;

    // ─────────────── DRYING SECTION — GROUP 2 ───────────────
    dryingSectionGroup2UpperMasterFaultAlarm         : BOOL;  // G2 Upper Master fault / trip
    dryingSectionGroup2UpperMasterCoolingFaultAlarm  : BOOL;  // G2 Upper Master forced cooling fault
    dryingSectionGroup2UpperSlave1FaultAlarm         : BOOL;  // G2 Upper Slave1 fault / trip
    dryingSectionGroup2UpperSlave1CoolingFaultAlarm  : BOOL;  // G2 Upper Slave1 forced cooling fault
    dryingSectionGroup2UpperSlave2FaultAlarm         : BOOL;  // G2 Upper Slave2 fault / trip
    dryingSectionGroup2UpperSlave2CoolingFaultAlarm  : BOOL;  // G2 Upper Slave2 forced cooling fault

    dryingSectionGroup2LowerMasterFaultAlarm         : BOOL;  // G2 Lower Master fault / trip
    dryingSectionGroup2LowerMasterCoolingFaultAlarm  : BOOL;  // G2 Lower Master forced cooling fault
    dryingSectionGroup2LowerSlave1FaultAlarm         : BOOL;  // G2 Lower Slave1 fault / trip
    dryingSectionGroup2LowerSlave1CoolingFaultAlarm  : BOOL;  // G2 Lower Slave1 forced cooling fault
    dryingSectionGroup2LowerSlave2FaultAlarm         : BOOL;  // G2 Lower Slave2 fault / trip
    dryingSectionGroup2LowerSlave2CoolingFaultAlarm  : BOOL;  // G2 Lower Slave2 forced cooling fault

    // ── FABRIC OVERRUN PROTECTION — GROUP 2 ───────────────────────────────────
    upperDryingSectionGroup2FabricOverrunOperatorSideAlarm : BOOL;  // Fabric overrun detected on operator side (sensor active)
    upperDryingSectionGroup2FabricOverrunDriveSideAlarm    : BOOL;  // Fabric overrun detected on drive side (sensor active)
    lowerDryingSectionGroup2FabricOverrunOperatorSideAlarm : BOOL;  // Fabric overrun detected on operator side (sensor active)
    lowerDryingSectionGroup2FabricOverrunDriveSideAlarm    : BOOL;  // Fabric overrun detected on drive side (sensor active)

    // ───────── DRYING SECTION — FABRIC STRETCHER — GROUP 2 ─────────
    upperDryingSectionGroup2FabricStretcherMotorFaultAlarm : BOOL;  // Upper fabric stretcher motor fault (G2)
    lowerDryingSectionGroup2FabricStretcherMotorFaultAlarm : BOOL;  // Lower fabric stretcher motor fault (G2)

    // ───────── DRYING SECTION — AUXILIARIES — GROUP 2 ─────────
    dryingSectionGroup2PickUpRollPosFaultAlarm       : BOOL;  // EN: G2 pick-up roll positioner fault / PT: Falha do posicionador do rolo pick-up G2
    dryingSectionGroup2BabyDryerScraperOscFaultAlarm : BOOL;  // EN: G2 babydryer scraper oscillator fault / PT: Falha do oscilador da raspa do babydryer G2
    dryingSectionGroup2UpperScraperOscFaultAlarm     : BOOL;  // EN: G2 upper group scraper oscillator fault / PT: Falha do oscilador da raspa do grupo superior G2
    dryingSectionGroup2LowerScraperOscFaultAlarm     : BOOL;  // EN: G2 lower group scraper oscillator fault / PT: Falha do oscilador da raspa do grupo inferior G2
	dryingSectionGroup2PaperBreakAlarm : BOOL;

    // ─────────────── DRYING SECTION — GROUP 3 ───────────────
    dryingSectionGroup3UpperMasterFaultAlarm         : BOOL;  // G3 Upper Master fault / trip
    dryingSectionGroup3UpperMasterCoolingFaultAlarm  : BOOL;  // G3 Upper Master forced cooling fault
    dryingSectionGroup3UpperSlave1FaultAlarm         : BOOL;  // G3 Upper Slave1 fault / trip
    dryingSectionGroup3UpperSlave1CoolingFaultAlarm  : BOOL;  // G3 Upper Slave1 forced cooling fault
    dryingSectionGroup3UpperSlave2FaultAlarm         : BOOL;  // G3 Upper Slave2 fault / trip
    dryingSectionGroup3UpperSlave2CoolingFaultAlarm  : BOOL;  // G3 Upper Slave2 forced cooling fault

    dryingSectionGroup3LowerMasterFaultAlarm         : BOOL;  // G3 Lower Master fault / trip
    dryingSectionGroup3LowerMasterCoolingFaultAlarm  : BOOL;  // G3 Lower Master forced cooling fault
    dryingSectionGroup3LowerSlave1FaultAlarm         : BOOL;  // G3 Lower Slave1 fault / trip
    dryingSectionGroup3LowerSlave1CoolingFaultAlarm  : BOOL;  // G3 Lower Slave1 forced cooling fault
    dryingSectionGroup3LowerSlave2FaultAlarm         : BOOL;  // G3 Lower Slave2 fault / trip
    dryingSectionGroup3LowerSlave2CoolingFaultAlarm  : BOOL;  // G3 Lower Slave2 forced cooling fault

    // ── FABRIC OVERRUN PROTECTION — GROUP 3 ───────────────────────────────────
    upperDryingSectionGroup3FabricOverrunOperatorSideAlarm : BOOL;  // Fabric overrun detected on operator side (sensor active)
    upperDryingSectionGroup3FabricOverrunDriveSideAlarm    : BOOL;  // Fabric overrun detected on drive side (sensor active)
    lowerDryingSectionGroup3FabricOverrunOperatorSideAlarm : BOOL;  // Fabric overrun detected on operator side (sensor active)
    lowerDryingSectionGroup3FabricOverrunDriveSideAlarm    : BOOL;  // Fabric overrun detected on drive side (sensor active)

    // ───────── DRYING SECTION — FABRIC STRETCHER — GROUP 3 ─────────
    upperDryingSectionGroup3FabricStretcherMotorFaultAlarm : BOOL;  // Upper fabric stretcher motor fault (G3)
    lowerDryingSectionGroup3FabricStretcherMotorFaultAlarm : BOOL;  // Lower fabric stretcher motor fault (G3)

    // ───────── DRYING SECTION — AUXILIARIES — GROUP 3 ─────────
    dryingSectionGroup3PickUpRollPosFaultAlarm       : BOOL;  // EN: G3 pick-up roll positioner fault / PT: Falha do posicionador do rolo pick-up G3
    dryingSectionGroup3BabyDryerScraperOscFaultAlarm : BOOL;  // EN: G3 babydryer scraper oscillator fault / PT: Falha do oscilador da raspa do babydryer G3
    dryingSectionGroup3UpperScraperOscFaultAlarm     : BOOL;  // EN: G3 upper group scraper oscillator fault / PT: Falha do oscilador da raspa do grupo superior G3
    dryingSectionGroup3LowerScraperOscFaultAlarm     : BOOL;  // EN: G3 lower group scraper oscillator fault / PT: Falha do oscilador da raspa do grupo inferior G3
	dryingSectionGroup3PaperBreakAlarm : BOOL;
    // ─────────────── CENTRIFUGAL PRESSURE SCREEN ───────────────
    cpsUnitFaultAlarm                        : BOOL;  // Screen unit fault / trip

    // ─────────────── COUCH PIT PUMP & MIXER ───────────────
    couchPitPumpFaultAlarm                   : BOOL;  // Couch pit pump fault / trip

    // ─────────────── WIRE PIT PUMP ───────────────
    wirePitPumpFaultAlarm                    : BOOL;  // Wire pit pump fault / trip

    // ─────────────── STOCK PUMP ───────────────
    stockPumpFaultAlarm                      : BOOL;  // Stock pump fault / trip

    // ─────────────── MIXING PUMP ───────────────
    mixingPumpFaultAlarm                     : BOOL;  // Mixing pump fault / trip

    // ─────────────── VACUUM PUMPS ───────────────
    vacuumPump1FaultAlarm                    : BOOL;  // Vacuum pump 1 fault / trip
    vacuumPump2FaultAlarm                    : BOOL;  // Vacuum pump 2 fault / trip

    // ─────────────── LOW VACUUM EXHAUST FAN ───────────────
    lowVacuumFanFaultAlarm                   : BOOL;  // Low vacuum exhaust fan fault / trip

    // ─────────────── LUBRIFICATION PUMPS ───────────────
    lubricationPump1FaultAlarm              : BOOL;  // Lubrication pump 1 fault / trip
    lubricationPump2FaultAlarm              : BOOL;  // Lubrication pump 2 fault / trip
    lubricationMinPressureFaultAlarm        : BOOL;  // Minimum pressure not reached / trip
    lubricationMaxPressureFaultAlarm        : BOOL;  // Overpressure in lubrication circuit / trip
	lubricationTankHighTemperatureAlarm 	: BOOL;
	lubricationCircuitHighTemperatureAlarm 	: BOOL;

END_STRUCT
END_TYPE

// ---- Function Blocks/Rewinder/DataTypes/Rewinder_TypePressRoll.TcDUT
TYPE Rewinder_TypePressRoll :
	STRUCT
			
		rollDiameter	: REAL := 0.00;			//Forming board manual speed (Slow speed)
		pressureSetpoint	: REAL := 0.00;			//Forming board manual speed (Slow speed)
				
	END_STRUCT
END_TYPE

// ---- Function Blocks/Rewinder/DataTypes/Rewinder_TypeBrakeControl.TcDUT
TYPE Rewinder_TypeBrakeControl :
	STRUCT
		
	
		rollDiameter		: REAL;			//Forming board manual speed (Slow speed)
		pressureSetpoint	: REAL;			//Forming board manual speed (Slow speed)
		tensionSetpoint		: REAL;
			
	END_STRUCT
END_TYPE

// ---- POUs/MAIN.TcPOU
PROGRAM MAIN
VAR
	instFB_DryingSectionLubrificationControl_V1 : FB_DryingSectionLubrificationControl_V1;
	instFB_SavePersistentData	: FB_SavePersistentData;
	instFB_SpeedDroopControlMst : FB_SpeedDroopControl_1;
	instFB_SpeedDroopControlSlv : FB_FormingBoardDriveControl;
	instFB_DryingSectionDriveControl_GR1 : FB_DryingSectionDriveControl_V1;
	instFB_DryingSectionDriveControl_GR2 : FB_DryingSectionDriveControl_V1;
	
	instFFB_PressSectionDriveControl_V1 : FB_PressSectionDriveControl_V2;
	
	                 

	FB_SoftstarterWithBypass_0: FB_SoftstarterWithBypass;
	FB_PressureControl_0: FB_PressureControl;
	FB_MixPumpControl_0: FB_MixPumpControl;
	FB_HeadboxLipsPWMControl_0: FB_HeadboxLipsPWMControl;
	instPWM: CTRL_PWM;
	instFB_MixPumpControl: FB_MixPumpControl;
	instFB_FormingBoardRollUpDown: FB_FormingBoardRollUpDown;
	instFB_HeadboxLipsPWMControl: FB_HeadboxLipsPWMControl;
	instFB_FormingBoarWireStrech: FB_FormingBoardRollUpDown;
	instFB_FormingBoardWireStretchControl: FB_FormingBoardWireStretchControl;
	instFB_SoftstarterSimpleCPS: FB_SimpleMotorStart_V2;
	// Centrifugal Pressure Screen (CPS) running (Depurador cabeçeira)
	CPSRunning: BOOL;
	instFB_LevelControlWirePit: FB_LevelControl_V2;
	instFB_LevelControlCouchPit: FB_LevelControl_V2;
	stop: BOOL;
	formingBoardWireLimitInibit: BOOL;
	instFB_SoftstarterSimpleCouchPitMixer: FB_SimpleMotorStart_V2;
	instFB_SoftstarterWithBypassFormingBoard: FB_SoftstarterWithBypass;
	instFB_SoftstarterWithBypassSuctionRoll: FB_SoftstarterWithBypass_V1;
	FB_SoftstarterWithBypassTest: FB_SoftstarterWithBypass;
	FB_SimpleMotorStart_V2_Test: FB_SimpleMotorStart_V2;
	instFB_SoftstarterWithBypass_V1: FB_SoftstarterWithBypass_V1;
	instFB_PressureControl_V1StockPumpC: FB_PressureControl_V1;
	instFB_SoftstarterWithBypass_FormingBoard: FB_SoftstarterWithBypass_V1;
	instFB_PressureControl_V1: FB_PressureControl_V1;
	instFB_FormingBoardDriveControl_V1: FB_FormingBoardControl_V1;
	instFB_MixPumpControl_V1: FB_MixPumpControl_V1;
	instFB_ProcessControlerStockPump: FB_VfdProcessControler;
	instFB_ProcessControlerWirePitPump: FB_WirePitControl;
	instFB_ValveProcessControlerWhiteWaterSilo : FB_ValveProcessControler;
	formingBoardNextGrReference: REAL;
	pressSectionNextGrReference: REAL;
	dryingSec1NextGrReference: REAL;
	dryingSec2NextGrReference: REAL;
	
	instFB_DryingSectionDriveControl_GR3: FB_DryingSectionDriveControl_V1;
	
	instFB_DryingSectionDriveControlV2_GR3: FB_DryingSectionDriveControl_V2;
	
	
	
	instFB_RewinderControl_V1 : FB_RewinderControl_V1;
	
	
	
	instFB_DryingSectionDriveControl_V3_GR1: FB_DryingSectionDriveControl_V3;
	instFB_DryingSectionDriveControl_V3_GR2: FB_DryingSectionDriveControl_V3;
	instFB_DryingSectionDriveControl_V3_GR3: FB_DryingSectionDriveControl_V3;
	
	
	initVariables : BOOL;
	rInitVariables : BOOL;
	initVariablesOld : BOOL;
	
	
	dryingSectionGr1NextGroupReference: REAL;
	dryingSectionGr2NextGroupReference: REAL;
	dryingSectionGr3NextGroupReference: REAL;
	instFB_SoftstarterWithBypassPress1: FB_SoftstarterWithBypass_V1;
	instFB_SoftstarterWithBypassPress2: FB_SoftstarterWithBypass_V1;
	bypassFault: BOOL;
	startNotAllowed: BOOL;
	instFB_WinderDriveControl_V1: FB_WinderDriveControl_V1;
	FB_FormingBoardControl_V3_0: FB_FormingBoardControl_V3;
	pressSectionNextGroupReference: REAL;
	
	
	firstScan	:BOOL := TRUE;
	
	
	vacumPumpSoftStartOK: BOOL;
	instTOFvacumPumpSoftstart: TOF;
	startSoftstartContactorFromPressFelt1: BOOL;
	startSoftstartFromPressFelt1: BOOL;
	startSoftstartContactorFromPressFelt2: BOOL;
	startSoftstartFromPressFelt2: BOOL;
	instFB_FB_SimpleMotorStart_V3_VaccumSealPump: FB_SimpleMotorStart_V3;
	instFB_FB_SimpleMotorStart_V3_lowVacuumExhaustFan: FB_SimpleMotorStart_V3;
	instFB_FB_SimpleMotorStart_V3_VaccumSeparator: FB_SimpleMotorStart_V3;
	instFB_FB_SimpleMotorStart_V3_FormingTailCutterNozzle: FB_SimpleMotorStart_V3;
	instFB_FB_SimpleMotorStart_V3_FormingWireShower: FB_SimpleMotorStart_V3;
	
	instFB_AlarmControl	: FB_AlarmControl;
	
	
	
//Write SDO
 fbSdoWrite : FB_EcCoESdoWrite;
    sNetId     : T_AmsNetId := '172.16.2.131.2.1'; (* NetId of EtherCAT Master *)
    nSlaveAddr : UINT := 1005; (* Port Number of EtherCAT Slave *)
    nIndex     : WORD := 16#4062; (* CoE Object Index *)
    nSubIndex  : BYTE := 1; (* Subindex of CoE Object *)
    nValue     : UINT := 2; (* variable to be written to the CoE Object *)
    bExecute   : BOOL; (* rising edge starts writing to the CoE Object *)
    bError     : BOOL;
    nErrId     : UDINT;
	
tractionRoll_speedSetpoint : UINT;
sctionRoll_speedSetpoint : UINT;

firstPress_speedSetpoint : UINT;
secondPress_speedSetpoint : UINT;

upperMaster_1GR_speedSetpoint : UINT;
upperSlave_1GR_speedSetpoint : UINT;
lowerMaster_1GR_speedSetpoint : UINT;

upperMaster_2GR_speedSetpoint : UINT;
upperSlave_2GR_speedSetpoint : UINT;
lowerMaster_2GR_speedSetpoint : UINT;
lowerSlave_2GR_speedSetpoint : UINT;

upperMaster_3GR_speedSetpoint : UINT;
upperSlave_3GR_speedSetpoint : UINT;
lowerMaster_3GR_speedSetpoint : UINT;
lowerSlave_3GR_speedSetpoint : UINT;

rewinder_speedSetpoint	 : UINT;
	
	adsWriteState: INT;
	instFB_ProcessControlerWirePitPumpTest: FB_WirePitControl_1;
END_VAR

//────────────────────────────────────────────
// READ I/O MODULES
//────────────────────────────────────────────

// UG I/O Modules
P1_100_UG01();
P1_100_UG02();
P1_100_UG03_SuctionRoll();
P1_100_UG04();
P1_100_UG05();
P1_300_UG06_TractionRoll();

// Digital Inputs
P1_050_DI1();
P1_050_DI2();
P1_050_DI3();
P9_050_DI1();
P9_050_DI2();
P9_050_DI3();
P10_050_DI1();
P10_050_DI2();
P10_050_DI3();
P10_050_DI4();
P10_050_DI5();
P10_050_DI6();
P10_050_DI7();
P10_050_DI8();

// Digital Outputs
P1_050_DO1();
P1_050_DO2();
P1_050_DO3();
P9_050_DO1();
P9_050_DO2();
P9_050_DO3();
P10_050_DO1();
P10_050_DO2();
P10_050_DO3();
P10_050_DO4();

// Analog Inputs
P1_050_AI1();
P1_050_AI2();
P1_050_AI3();
P1_050_AI4();
P9_050_AI1();
P10_050_AI1();
P10_050_AI2();

// Analog Outputs
P1_050_AQ1();
P1_050_AQ2();
P10_050_AO1();


CP1_050_DI1();
CP1_050_DO1();
CP1_050_AO1();


// Safety PLC
P1_050_SP1();

//────────────────────────────────────────────
// READ DRIVES
//────────────────────────────────────────────

// Press Section
P11_400_UG01_SecondPress();     // Second Press
P12_400_UG01_FirstPress();      // First Press

// Drying Section — Group 1
P13_500_UG01_1GR_UpperSlave();  // Group 1 - Upper Slave
P13_500_UG02_1GR_LowerMaster(); // Group 1 - Lower Master
P13_500_UG03_1GR_UpperMaster(); // Group 1 - Upper Master

// Drying Section — Group 2
P13_501_UG01_2GR_LowerSlave();  // Group 2 - Lower Slave
P13_501_UG02_2GR_UpperSlave();  // Group 2 - Upper Slave
P13_501_UG03_2GR_LowerMaster(); // Group 2 - Lower Master
P14_501_UG01_2GR_UpperMaster(); // Group 2 - Upper Master

// Drying Section — Group 3
P14_502_UG01_3GR_LowerSlave();  // Group 3 - Lower Slave
P14_502_UG02_3GR_UpperSlave();  // Group 3 - Upper Slave
P14_502_UG03_3GR_LowerMaster(); // Group 3 - Lower Master
P14_502_UG04_3GR_UpperMaster(); // Group 3 - Upper Master

//Winder group
P15_600_UG01_Rewinder();
//────────────────────────────────────────────
// PROGRAM FUNCTION BLOCK CALLS
//────────────────────────────────────────────

// Forming Section
_100_FormingBoardControl();
_110_FormingBoardAux();

// Press Section
_200_PressSectionControl();

// Drying Section
_500_DryingSectionGroup1DriveControl();
_501_DryingSectionGroup2DriveControl();
_502_DryingSectionGroup3DriveControl();
_550_DryingSectionLubrification();
_600_WinderGroup();

_888_Alarms();


// Headbox / Stock Prep / Wet End Auxiliary Systems
//_HeadBoxAuxiliaryControls();
_MixPumpControl_1();
_WirePitControl();
_CentrifugalPressureScreenControl();
_CouchPitPumpControl();
_CouchPitMixerControl();
_VaccumPumps();
//_StockPumpControl();
_StockPumpControl_1();

// Testing & Debug
_FunctionBlockTest();

//────────────────────────────────────────────
// SYSTEM MANAGEMENT
//────────────────────────────────────────────

// Save persistent variables to CPU
instFB_SavePersistentData();

// Enable Safety PLC
P1_050_SP1.run := TRUE;

// Perform machine-wide reset
machineReset();


rInitVariables := initVariables AND NOT initVariablesOld;

IF rInitVariables THEN
	
	_000_Init_Variables();

END_IF

initVariablesOld := initVariables;



IF firstScan THEN
	
	_001_FirstScan();

END_IF


sctionRoll_speedSetpoint:= (P1_100_UG03_SuctionRoll.pdoSpeedSet); //Address 1021
tractionRoll_speedSetpoint := (P1_300_UG06_TractionRoll.pdoSpeedSet); //Addres 1024

secondPress_speedSetpoint := (P11_400_UG01_SecondPress.pdoSpeedSet); //1052
firstPress_speedSetpoint := (P12_400_UG01_FirstPress.pdoSpeedSet); //1053

upperSlave_1GR_speedSetpoint := (P13_500_UG01_1GR_UpperSlave.pdoSpeedSet); //1054
lowerMaster_1GR_speedSetpoint := (P13_500_UG02_1GR_LowerMaster.pdoSpeedSet);//1055
upperMaster_1GR_speedSetpoint := (P13_500_UG03_1GR_UpperMaster.pdoSpeedSet);//1056

lowerSlave_2GR_speedSetpoint:= (P13_501_UG01_2GR_LowerSlave.pdoSpeedSet);//1057
upperSlave_2GR_speedSetpoint:= (P13_501_UG02_2GR_UpperSlave.pdoSpeedSet);//1058
lowerMaster_2GR_speedSetpoint:= (P13_501_UG03_2GR_LowerMaster.pdoSpeedSet);//1059
upperMaster_2GR_speedSetpoint:= (P14_501_UG01_2GR_UpperMaster.pdoSpeedSet);//1060

lowerSlave_3GR_speedSetpoint:= (P14_502_UG01_3GR_LowerSlave.pdoSpeedSet);//1061
upperSlave_3GR_speedSetpoint:= (P14_502_UG02_3GR_UpperSlave.pdoSpeedSet);//1062
lowerMaster_3GR_speedSetpoint:= (P14_502_UG03_3GR_LowerMaster.pdoSpeedSet);//1063
upperMaster_3GR_speedSetpoint:= (P14_502_UG04_3GR_UpperMaster.pdoSpeedSet);//1064

rewinder_speedSetpoint:= (P15_600_UG01_Rewinder.pdoSpeedSet);//1065

// NOTE:
// - You had duplicated CASE label "2:" twice. The second one must be "3:" (1053).
// - Below continues the sequence following your exact pattern.


bExecute := TRUE;

CASE adsWriteState OF

    0:
        fbSdoWrite(
            sNetId     := '192.168.100.1.3.1',
            nSlaveAddr := 1021,
            nIndex     := 16#3004,
            nSubIndex  := 1,
            pSrcBuf    := ADR(sctionRoll_speedSetpoint),
            cbBufLen   := SIZEOF(sctionRoll_speedSetpoint),
            bExecute   := bExecute
        );

        IF NOT fbSdoWrite.bBusy THEN
            bExecute := FALSE;
            IF NOT fbSdoWrite.bError THEN
                bError := FALSE;
                nErrId := 0;
                adsWriteState := adsWriteState + 1;
            ELSE
                bError := fbSdoWrite.bError;
                nErrId := fbSdoWrite.nErrId;
                adsWriteState := adsWriteState + 1;
				
            END_IF

            fbSdoWrite(bExecute := FALSE);
        END_IF

    1:
        fbSdoWrite(
            sNetId     := '192.168.100.1.3.1',
            nSlaveAddr := 1024,
            nIndex     := 16#3004,
            nSubIndex  := 1,
            pSrcBuf    := ADR(tractionRoll_speedSetpoint),
            cbBufLen   := SIZEOF(tractionRoll_speedSetpoint),
            bExecute   := bExecute
        );

        IF NOT fbSdoWrite.bBusy THEN
            bExecute := FALSE;
            IF NOT fbSdoWrite.bError THEN
                bError := FALSE;
                nErrId := 0;
                adsWriteState := adsWriteState + 1;
            ELSE
                bError := fbSdoWrite.bError;
                nErrId := fbSdoWrite.nErrId;
                adsWriteState := adsWriteState + 1;
				
            END_IF

            fbSdoWrite(bExecute := FALSE);
        END_IF

    2:
        fbSdoWrite(
            sNetId     := '192.168.100.1.3.1',
            nSlaveAddr := 1052,
            nIndex     := 16#3004,
            nSubIndex  := 1,
            pSrcBuf    := ADR(secondPress_speedSetpoint),
            cbBufLen   := SIZEOF(secondPress_speedSetpoint),
            bExecute   := bExecute
        );

        IF NOT fbSdoWrite.bBusy THEN
            bExecute := FALSE;
            IF NOT fbSdoWrite.bError THEN
                bError := FALSE;
                nErrId := 0;
                adsWriteState := adsWriteState + 1;
            ELSE
                bError := fbSdoWrite.bError;
                nErrId := fbSdoWrite.nErrId;
                adsWriteState := adsWriteState + 1;
				
            END_IF

            fbSdoWrite(bExecute := FALSE);
        END_IF

    3: // was duplicated as "2:" in your snippet
        fbSdoWrite(
            sNetId     := '192.168.100.1.3.1',
            nSlaveAddr := 1053,
            nIndex     := 16#3004,
            nSubIndex  := 1,
            pSrcBuf    := ADR(firstPress_speedSetpoint),
            cbBufLen   := SIZEOF(firstPress_speedSetpoint),
            bExecute   := bExecute
        );

        IF NOT fbSdoWrite.bBusy THEN
            bExecute := FALSE;
            IF NOT fbSdoWrite.bError THEN
                bError := FALSE;
                nErrId := 0;
                adsWriteState := adsWriteState + 1;
            ELSE
                bError := fbSdoWrite.bError;
                nErrId := fbSdoWrite.nErrId;
                adsWriteState := adsWriteState + 1;
				
            END_IF

            fbSdoWrite(bExecute := FALSE);
        END_IF

    4:
        fbSdoWrite(
            sNetId     := '192.168.100.1.3.1',
            nSlaveAddr := 1054,
            nIndex     := 16#3004,
            nSubIndex  := 1,
            pSrcBuf    := ADR(upperSlave_1GR_speedSetpoint),
            cbBufLen   := SIZEOF(upperSlave_1GR_speedSetpoint),
            bExecute   := bExecute
        );

        IF NOT fbSdoWrite.bBusy THEN
            bExecute := FALSE;
            IF NOT fbSdoWrite.bError THEN
                bError := FALSE;
                nErrId := 0;
                adsWriteState := adsWriteState + 1;
            ELSE
                bError := fbSdoWrite.bError;
                nErrId := fbSdoWrite.nErrId;
                adsWriteState := adsWriteState + 1;
				
            END_IF

            fbSdoWrite(bExecute := FALSE);
        END_IF

    5:
        fbSdoWrite(
            sNetId     := '192.168.100.1.3.1',
            nSlaveAddr := 1055,
            nIndex     := 16#3004,
            nSubIndex  := 1,
            pSrcBuf    := ADR(lowerMaster_1GR_speedSetpoint),
            cbBufLen   := SIZEOF(lowerMaster_1GR_speedSetpoint),
            bExecute   := bExecute
        );

        IF NOT fbSdoWrite.bBusy THEN
            bExecute := FALSE;
            IF NOT fbSdoWrite.bError THEN
                bError := FALSE;
                nErrId := 0;
                adsWriteState := adsWriteState + 1;
            ELSE
                bError := fbSdoWrite.bError;
                nErrId := fbSdoWrite.nErrId;
                adsWriteState := adsWriteState + 1;
				
            END_IF

            fbSdoWrite(bExecute := FALSE);
        END_IF

    6:
        fbSdoWrite(
            sNetId     := '192.168.100.1.3.1',
            nSlaveAddr := 1056,
            nIndex     := 16#3004,
            nSubIndex  := 1,
            pSrcBuf    := ADR(upperMaster_1GR_speedSetpoint),
            cbBufLen   := SIZEOF(upperMaster_1GR_speedSetpoint),
            bExecute   := bExecute
        );

        IF NOT fbSdoWrite.bBusy THEN
            bExecute := FALSE;
            IF NOT fbSdoWrite.bError THEN
                bError := FALSE;
                nErrId := 0;
                adsWriteState := adsWriteState + 1;
            ELSE
                bError := fbSdoWrite.bError;
                nErrId := fbSdoWrite.nErrId;
                adsWriteState := adsWriteState + 1;
				
            END_IF

            fbSdoWrite(bExecute := FALSE);
        END_IF

    7:
        fbSdoWrite(
            sNetId     := '192.168.100.1.3.1',
            nSlaveAddr := 1057,
            nIndex     := 16#3004,
            nSubIndex  := 1,
            pSrcBuf    := ADR(lowerSlave_2GR_speedSetpoint),
            cbBufLen   := SIZEOF(lowerSlave_2GR_speedSetpoint),
            bExecute   := bExecute
        );

        IF NOT fbSdoWrite.bBusy THEN
            bExecute := FALSE;
            IF NOT fbSdoWrite.bError THEN
                bError := FALSE;
                nErrId := 0;
                adsWriteState := adsWriteState + 1;
            ELSE
                bError := fbSdoWrite.bError;
                nErrId := fbSdoWrite.nErrId;
                adsWriteState := adsWriteState + 1;

				
            END_IF

            fbSdoWrite(bExecute := FALSE);
        END_IF

    8:
        fbSdoWrite(
            sNetId     := '192.168.100.1.3.1',
            nSlaveAddr := 1058,
            nIndex     := 16#3004,
            nSubIndex  := 1,
            pSrcBuf    := ADR(upperSlave_2GR_speedSetpoint),
            cbBufLen   := SIZEOF(upperSlave_2GR_speedSetpoint),
            bExecute   := bExecute
        );

        IF NOT fbSdoWrite.bBusy THEN
            bExecute := FALSE;
            IF NOT fbSdoWrite.bError THEN
                bError := FALSE;
                nErrId := 0;
                adsWriteState := adsWriteState + 1;
            ELSE
                bError := fbSdoWrite.bError;
                nErrId := fbSdoWrite.nErrId;
                adsWriteState := adsWriteState + 1;

				
            END_IF

            fbSdoWrite(bExecute := FALSE);
        END_IF

    9:
        fbSdoWrite(
            sNetId     := '192.168.100.1.3.1',
            nSlaveAddr := 1059,
            nIndex     := 16#3004,
            nSubIndex  := 1,
            pSrcBuf    := ADR(lowerMaster_2GR_speedSetpoint),
            cbBufLen   := SIZEOF(lowerMaster_2GR_speedSetpoint),
            bExecute   := bExecute
        );

        IF NOT fbSdoWrite.bBusy THEN
            bExecute := FALSE;
            IF NOT fbSdoWrite.bError THEN
                bError := FALSE;
                nErrId := 0;
                adsWriteState := adsWriteState + 1;
            ELSE
                bError := fbSdoWrite.bError;
                nErrId := fbSdoWrite.nErrId;
                adsWriteState := adsWriteState + 1;

				
            END_IF

            fbSdoWrite(bExecute := FALSE);
        END_IF

    10:
        fbSdoWrite(
            sNetId     := '192.168.100.1.3.1',
            nSlaveAddr := 1060,
            nIndex     := 16#3004,
            nSubIndex  := 1,
            pSrcBuf    := ADR(upperMaster_2GR_speedSetpoint),
            cbBufLen   := SIZEOF(upperMaster_2GR_speedSetpoint),
            bExecute   := bExecute
        );

        IF NOT fbSdoWrite.bBusy THEN
            bExecute := FALSE;
            IF NOT fbSdoWrite.bError THEN
                bError := FALSE;
                nErrId := 0;
                adsWriteState := adsWriteState + 1;
            ELSE
                bError := fbSdoWrite.bError;
                nErrId := fbSdoWrite.nErrId;
                adsWriteState := adsWriteState + 1;

				
            END_IF

            fbSdoWrite(bExecute := FALSE);
        END_IF

    11:
        fbSdoWrite(
            sNetId     := '192.168.100.1.3.1',
            nSlaveAddr := 1061,
            nIndex     := 16#3004,
            nSubIndex  := 1,
            pSrcBuf    := ADR(lowerSlave_3GR_speedSetpoint),
            cbBufLen   := SIZEOF(lowerSlave_3GR_speedSetpoint),
            bExecute   := bExecute
        );

        IF NOT fbSdoWrite.bBusy THEN
            bExecute := FALSE;
            IF NOT fbSdoWrite.bError THEN
                bError := FALSE;
                nErrId := 0;
                adsWriteState := adsWriteState + 1;
            ELSE
                bError := fbSdoWrite.bError;
                nErrId := fbSdoWrite.nErrId;
                adsWriteState := adsWriteState + 1;

				
            END_IF

            fbSdoWrite(bExecute := FALSE);
        END_IF

    12:
        fbSdoWrite(
            sNetId     := '192.168.100.1.3.1',
            nSlaveAddr := 1062,
            nIndex     := 16#3004,
            nSubIndex  := 1,
            pSrcBuf    := ADR(upperSlave_3GR_speedSetpoint),
            cbBufLen   := SIZEOF(upperSlave_3GR_speedSetpoint),
            bExecute   := bExecute
        );

        IF NOT fbSdoWrite.bBusy THEN
            bExecute := FALSE;
            IF NOT fbSdoWrite.bError THEN
                bError := FALSE;
                nErrId := 0;
                adsWriteState := adsWriteState + 1;
            ELSE
                bError := fbSdoWrite.bError;
                nErrId := fbSdoWrite.nErrId;
                adsWriteState := adsWriteState + 1;
;
				
            END_IF

            fbSdoWrite(bExecute := FALSE);
        END_IF

    13:
        fbSdoWrite(
            sNetId     := '192.168.100.1.3.1',
            nSlaveAddr := 1063,
            nIndex     := 16#3004,
            nSubIndex  := 1,
            pSrcBuf    := ADR(lowerMaster_3GR_speedSetpoint),
            cbBufLen   := SIZEOF(lowerMaster_3GR_speedSetpoint),
            bExecute   := bExecute
        );

        IF NOT fbSdoWrite.bBusy THEN
            bExecute := FALSE;
            IF NOT fbSdoWrite.bError THEN
                bError := FALSE;
                nErrId := 0;
                adsWriteState := adsWriteState + 1;
            ELSE
                bError := fbSdoWrite.bError;
                nErrId := fbSdoWrite.nErrId;
                adsWriteState := adsWriteState + 1;

				
            END_IF

            fbSdoWrite(bExecute := FALSE);
        END_IF

    14:
        fbSdoWrite(
            sNetId     := '192.168.100.1.3.1',
            nSlaveAddr := 1064,
            nIndex     := 16#3004,
            nSubIndex  := 1,
            pSrcBuf    := ADR(upperMaster_3GR_speedSetpoint),
            cbBufLen   := SIZEOF(upperMaster_3GR_speedSetpoint),
            bExecute   := bExecute
        );

        IF NOT fbSdoWrite.bBusy THEN
            bExecute := FALSE;
            IF NOT fbSdoWrite.bError THEN
                bError := FALSE;
                nErrId := 0;
                adsWriteState := adsWriteState + 1;
            ELSE
                bError := fbSdoWrite.bError;
                nErrId := fbSdoWrite.nErrId;
                adsWriteState := adsWriteState + 1;

				
            END_IF

            fbSdoWrite(bExecute := FALSE);
        END_IF

    15:
        fbSdoWrite(
            sNetId     := '192.168.100.1.3.1',
            nSlaveAddr := 1065,
            nIndex     := 16#3004,
            nSubIndex  := 1,
            pSrcBuf    := ADR(rewinder_speedSetpoint),
            cbBufLen   := SIZEOF(rewinder_speedSetpoint),
            bExecute   := bExecute
        );

        IF NOT fbSdoWrite.bBusy THEN
            bExecute := FALSE;
            IF NOT fbSdoWrite.bError THEN
                bError := FALSE;
                nErrId := 0;
                adsWriteState := 0; // moves to 16
            ELSE
                bError := fbSdoWrite.bError;
                nErrId := fbSdoWrite.nErrId;
                adsWriteState := 0;

            END_IF

            fbSdoWrite(bExecute := FALSE);
        END_IF


END_CASE

METHOD _000_Init_Variables
VAR_INPUT
END_VAR

P1_300_UG06_TractionRoll.deviceConfig.MotorSpeedInputLow := 0.0;
P1_300_UG06_TractionRoll.deviceConfig.MotorSpeedInputHigh := 360.4;
P1_300_UG06_TractionRoll.deviceConfig.MotorSpeedOutputLow := 0.0;
P1_300_UG06_TractionRoll.deviceConfig.MotorSpeedOutputHigh := 360.4;
P1_300_UG06_TractionRoll.deviceConfig.speedSetpointInputLow := 0.0;
P1_300_UG06_TractionRoll.deviceConfig.speedSetpointInputHigh := 360.4;
P1_300_UG06_TractionRoll.deviceConfig.speedSetpointOutputLow := 0.0;
P1_300_UG06_TractionRoll.deviceConfig.speedSetpointOutputHigh := 360.4;


P1_100_UG03_SuctionRoll.deviceConfig.MotorSpeedInputLow := 0.0;
P1_100_UG03_SuctionRoll.deviceConfig.MotorSpeedInputHigh := 329.3;
P1_100_UG03_SuctionRoll.deviceConfig.MotorSpeedOutputLow := 0.0;
P1_100_UG03_SuctionRoll.deviceConfig.MotorSpeedOutputHigh := 329.3;
P1_100_UG03_SuctionRoll.deviceConfig.speedSetpointInputLow := 0.0;
P1_100_UG03_SuctionRoll.deviceConfig.speedSetpointInputHigh := 329.3;
P1_100_UG03_SuctionRoll.deviceConfig.speedSetpointOutputLow := 0.0;
P1_100_UG03_SuctionRoll.deviceConfig.speedSetpointOutputHigh := 329.3;
//Torque Enable
P1_100_UG03_SuctionRoll.deviceConfig.torqueLimiterEnabled := TRUE;
P1_100_UG03_SuctionRoll.deviceConfig.operationMode := 4;



P11_400_UG01_SecondPress.deviceConfig.MotorSpeedInputLow := 0.0;
P11_400_UG01_SecondPress.deviceConfig.MotorSpeedInputHigh := 374;
P11_400_UG01_SecondPress.deviceConfig.MotorSpeedOutputLow := 0.0;
P11_400_UG01_SecondPress.deviceConfig.MotorSpeedOutputHigh := 374;
P11_400_UG01_SecondPress.deviceConfig.speedSetpointInputLow := 0.0;
P11_400_UG01_SecondPress.deviceConfig.speedSetpointInputHigh := 374;
P11_400_UG01_SecondPress.deviceConfig.speedSetpointOutputLow := 0.0;
P11_400_UG01_SecondPress.deviceConfig.speedSetpointOutputHigh := 374;


P12_400_UG01_FirstPress.deviceConfig.MotorSpeedInputLow := 0.0;
P12_400_UG01_FirstPress.deviceConfig.MotorSpeedInputHigh := 239.9;
P12_400_UG01_FirstPress.deviceConfig.MotorSpeedOutputLow := 0.0;
P12_400_UG01_FirstPress.deviceConfig.MotorSpeedOutputHigh := 239.9;
P12_400_UG01_FirstPress.deviceConfig.speedSetpointInputLow := 0.0;
P12_400_UG01_FirstPress.deviceConfig.speedSetpointInputHigh := 239.9;
P12_400_UG01_FirstPress.deviceConfig.speedSetpointOutputLow := 0.0;
P12_400_UG01_FirstPress.deviceConfig.speedSetpointOutputHigh := 239.9;
//Torque Enable
P12_400_UG01_FirstPress.deviceConfig.torqueLimiterEnabled := TRUE;
P12_400_UG01_FirstPress.deviceConfig.operationMode := 4;



//============================
// DRYING SECTION — GROUP 1
//============================

// Upper Slave
P13_500_UG01_1GR_UpperSlave.deviceConfig.MotorSpeedInputLow := 0.0;
P13_500_UG01_1GR_UpperSlave.deviceConfig.MotorSpeedInputHigh := 750;
P13_500_UG01_1GR_UpperSlave.deviceConfig.MotorSpeedOutputLow := 0.0;
P13_500_UG01_1GR_UpperSlave.deviceConfig.MotorSpeedOutputHigh := 750;
P13_500_UG01_1GR_UpperSlave.deviceConfig.speedSetpointInputLow := 0.0;
P13_500_UG01_1GR_UpperSlave.deviceConfig.speedSetpointInputHigh := 750;
P13_500_UG01_1GR_UpperSlave.deviceConfig.speedSetpointOutputLow := 0.0;
P13_500_UG01_1GR_UpperSlave.deviceConfig.speedSetpointOutputHigh := 750;
P13_500_UG01_1GR_UpperSlave.deviceConfig.torqueLimiterEnabled := TRUE;
P13_500_UG01_1GR_UpperSlave.deviceConfig.operationMode := 4;

// Lower Master
P13_500_UG02_1GR_LowerMaster.deviceConfig.MotorSpeedInputLow := 0.0;
P13_500_UG02_1GR_LowerMaster.deviceConfig.MotorSpeedInputHigh := 750;
P13_500_UG02_1GR_LowerMaster.deviceConfig.MotorSpeedOutputLow := 0.0;
P13_500_UG02_1GR_LowerMaster.deviceConfig.MotorSpeedOutputHigh := 750;
P13_500_UG02_1GR_LowerMaster.deviceConfig.speedSetpointInputLow := 0.0;
P13_500_UG02_1GR_LowerMaster.deviceConfig.speedSetpointInputHigh := 750;
P13_500_UG02_1GR_LowerMaster.deviceConfig.speedSetpointOutputLow := 0.0;
P13_500_UG02_1GR_LowerMaster.deviceConfig.speedSetpointOutputHigh := 750;
//P13_500_UG02_1GR_LowerMaster.deviceConfig.torqueLimiterEnabled := FALSE;
//P13_500_UG02_1GR_LowerMaster.deviceConfig.operationMode := 4;

// Upper Master
P13_500_UG03_1GR_UpperMaster.deviceConfig.MotorSpeedInputLow := 0.0;
P13_500_UG03_1GR_UpperMaster.deviceConfig.MotorSpeedInputHigh := 750;
P13_500_UG03_1GR_UpperMaster.deviceConfig.MotorSpeedOutputLow := 0.0;
P13_500_UG03_1GR_UpperMaster.deviceConfig.MotorSpeedOutputHigh := 750;
P13_500_UG03_1GR_UpperMaster.deviceConfig.speedSetpointInputLow := 0.0;
P13_500_UG03_1GR_UpperMaster.deviceConfig.speedSetpointInputHigh := 750;
P13_500_UG03_1GR_UpperMaster.deviceConfig.speedSetpointOutputLow := 0.0;
P13_500_UG03_1GR_UpperMaster.deviceConfig.speedSetpointOutputHigh := 750;
//P13_500_UG03_1GR_UpperMaster.deviceConfig.torqueLimiterEnabled := FALSE;
//P13_500_UG03_1GR_UpperMaster.deviceConfig.operationMode := 4;


//============================
// DRYING SECTION — GROUP 2
//============================

// Lower Slave
P13_501_UG01_2GR_LowerSlave.deviceConfig.MotorSpeedInputLow := 0.0;
P13_501_UG01_2GR_LowerSlave.deviceConfig.MotorSpeedInputHigh := 750;
P13_501_UG01_2GR_LowerSlave.deviceConfig.MotorSpeedOutputLow := 0.0;
P13_501_UG01_2GR_LowerSlave.deviceConfig.MotorSpeedOutputHigh := 750;
P13_501_UG01_2GR_LowerSlave.deviceConfig.speedSetpointInputLow := 0.0;
P13_501_UG01_2GR_LowerSlave.deviceConfig.speedSetpointInputHigh := 750;
P13_501_UG01_2GR_LowerSlave.deviceConfig.speedSetpointOutputLow := 0.0;
P13_501_UG01_2GR_LowerSlave.deviceConfig.speedSetpointOutputHigh := 750;
P13_501_UG01_2GR_LowerSlave.deviceConfig.torqueLimiterEnabled := TRUE;
P13_501_UG01_2GR_LowerSlave.deviceConfig.operationMode := 4;

// Upper Slave
P13_501_UG02_2GR_UpperSlave.deviceConfig.MotorSpeedInputLow := 0.0;
P13_501_UG02_2GR_UpperSlave.deviceConfig.MotorSpeedInputHigh := 750;
P13_501_UG02_2GR_UpperSlave.deviceConfig.MotorSpeedOutputLow := 0.0;
P13_501_UG02_2GR_UpperSlave.deviceConfig.MotorSpeedOutputHigh := 750;
P13_501_UG02_2GR_UpperSlave.deviceConfig.speedSetpointInputLow := 0.0;
P13_501_UG02_2GR_UpperSlave.deviceConfig.speedSetpointInputHigh := 750;
P13_501_UG02_2GR_UpperSlave.deviceConfig.speedSetpointOutputLow := 0.0;
P13_501_UG02_2GR_UpperSlave.deviceConfig.speedSetpointOutputHigh := 750;
P13_501_UG02_2GR_UpperSlave.deviceConfig.torqueLimiterEnabled := TRUE;
P13_501_UG02_2GR_UpperSlave.deviceConfig.operationMode := 4;

// Lower Master
P13_501_UG03_2GR_LowerMaster.deviceConfig.MotorSpeedInputLow := 0.0;
P13_501_UG03_2GR_LowerMaster.deviceConfig.MotorSpeedInputHigh := 750;
P13_501_UG03_2GR_LowerMaster.deviceConfig.MotorSpeedOutputLow := 0.0;
P13_501_UG03_2GR_LowerMaster.deviceConfig.MotorSpeedOutputHigh := 750;
P13_501_UG03_2GR_LowerMaster.deviceConfig.speedSetpointInputLow := 0.0;
P13_501_UG03_2GR_LowerMaster.deviceConfig.speedSetpointInputHigh := 750;
P13_501_UG03_2GR_LowerMaster.deviceConfig.speedSetpointOutputLow := 0.0;
P13_501_UG03_2GR_LowerMaster.deviceConfig.speedSetpointOutputHigh := 750;
//P13_501_UG03_2GR_LowerMaster.deviceConfig.torqueLimiterEnabled := FALSE;
//P13_501_UG03_2GR_LowerMaster.deviceConfig.operationMode := 4;

// Upper Master
P14_501_UG01_2GR_UpperMaster.deviceConfig.MotorSpeedInputLow := 0.0;
P14_501_UG01_2GR_UpperMaster.deviceConfig.MotorSpeedInputHigh := 750;
P14_501_UG01_2GR_UpperMaster.deviceConfig.MotorSpeedOutputLow := 0.0;
P14_501_UG01_2GR_UpperMaster.deviceConfig.MotorSpeedOutputHigh := 750;
P14_501_UG01_2GR_UpperMaster.deviceConfig.speedSetpointInputLow := 0.0;
P14_501_UG01_2GR_UpperMaster.deviceConfig.speedSetpointInputHigh := 750;
P14_501_UG01_2GR_UpperMaster.deviceConfig.speedSetpointOutputLow := 0.0;
P14_501_UG01_2GR_UpperMaster.deviceConfig.speedSetpointOutputHigh := 750;
//P14_501_UG01_2GR_UpperMaster.deviceConfig.torqueLimiterEnabled := FALSE;
//P14_501_UG01_2GR_UpperMaster.deviceConfig.operationMode := 4;


//============================
// DRYING SECTION — GROUP 3
//============================

// Lower Slave
P14_502_UG01_3GR_LowerSlave.deviceConfig.MotorSpeedInputLow := 0.0;
P14_502_UG01_3GR_LowerSlave.deviceConfig.MotorSpeedInputHigh := 750;
P14_502_UG01_3GR_LowerSlave.deviceConfig.MotorSpeedOutputLow := 0.0;
P14_502_UG01_3GR_LowerSlave.deviceConfig.MotorSpeedOutputHigh := 750;
P14_502_UG01_3GR_LowerSlave.deviceConfig.speedSetpointInputLow := 0.0;
P14_502_UG01_3GR_LowerSlave.deviceConfig.speedSetpointInputHigh := 750;
P14_502_UG01_3GR_LowerSlave.deviceConfig.speedSetpointOutputLow := 0.0;
P14_502_UG01_3GR_LowerSlave.deviceConfig.speedSetpointOutputHigh := 750;
P14_502_UG01_3GR_LowerSlave.deviceConfig.torqueLimiterEnabled := TRUE;
P14_502_UG01_3GR_LowerSlave.deviceConfig.operationMode := 4;

// Upper Slave
P14_502_UG02_3GR_UpperSlave.deviceConfig.MotorSpeedInputLow := 0.0;
P14_502_UG02_3GR_UpperSlave.deviceConfig.MotorSpeedInputHigh := 750;
P14_502_UG02_3GR_UpperSlave.deviceConfig.MotorSpeedOutputLow := 0.0;
P14_502_UG02_3GR_UpperSlave.deviceConfig.MotorSpeedOutputHigh := 750;
P14_502_UG02_3GR_UpperSlave.deviceConfig.speedSetpointInputLow := 0.0;
P14_502_UG02_3GR_UpperSlave.deviceConfig.speedSetpointInputHigh := 750;
P14_502_UG02_3GR_UpperSlave.deviceConfig.speedSetpointOutputLow := 0.0;
P14_502_UG02_3GR_UpperSlave.deviceConfig.speedSetpointOutputHigh := 750;
P14_502_UG02_3GR_UpperSlave.deviceConfig.torqueLimiterEnabled := TRUE;
P14_502_UG02_3GR_UpperSlave.deviceConfig.operationMode := 4;

// Lower Master
P14_502_UG03_3GR_LowerMaster.deviceConfig.MotorSpeedInputLow := 0.0;
P14_502_UG03_3GR_LowerMaster.deviceConfig.MotorSpeedInputHigh := 750;
P14_502_UG03_3GR_LowerMaster.deviceConfig.MotorSpeedOutputLow := 0.0;
P14_502_UG03_3GR_LowerMaster.deviceConfig.MotorSpeedOutputHigh := 750;
P14_502_UG03_3GR_LowerMaster.deviceConfig.speedSetpointInputLow := 0.0;
P14_502_UG03_3GR_LowerMaster.deviceConfig.speedSetpointInputHigh := 750;
P14_502_UG03_3GR_LowerMaster.deviceConfig.speedSetpointOutputLow := 0.0;
P14_502_UG03_3GR_LowerMaster.deviceConfig.speedSetpointOutputHigh := 750;
//P14_502_UG03_3GR_LowerMaster.deviceConfig.torqueLimiterEnabled := FALSE;
//P14_502_UG03_3GR_LowerMaster.deviceConfig.operationMode := 4;

// Upper Master
P14_502_UG04_3GR_UpperMaster.deviceConfig.MotorSpeedInputLow := 0.0;
P14_502_UG04_3GR_UpperMaster.deviceConfig.MotorSpeedInputHigh := 750;
P14_502_UG04_3GR_UpperMaster.deviceConfig.MotorSpeedOutputLow := 0.0;
P14_502_UG04_3GR_UpperMaster.deviceConfig.MotorSpeedOutputHigh := 750;
P14_502_UG04_3GR_UpperMaster.deviceConfig.speedSetpointInputLow := 0.0;
P14_502_UG04_3GR_UpperMaster.deviceConfig.speedSetpointInputHigh := 750;
P14_502_UG04_3GR_UpperMaster.deviceConfig.speedSetpointOutputLow := 0.0;
P14_502_UG04_3GR_UpperMaster.deviceConfig.speedSetpointOutputHigh := 750;
//P14_502_UG04_3GR_UpperMaster.deviceConfig.torqueLimiterEnabled := FALSE;
//P14_502_UG04_3GR_UpperMaster.deviceConfig.operationMode := 4;
END_METHOD

METHOD _001_FirstScan
VAR_INPUT
END_VAR

(*

paperMachineHmiCommands.dryingSectionGroup1SteamPressureAutoMan := FALSE;

	dryingSectionGroup1SteamPressureAutoSetpoint : REAL;  // Recovery speed increment [m/min or %] (Incremento de recuperação Grupo 1)
	dryingSectionGroup1SteamPressureManualSetpoint : REAL;  // Recovery speed increment [m/min or %] (Incremento de recuperação Grupo 1)
	
*)



paperMachineHmiCommands.dryingSectionGroup1SteamPressureAutoMan := FALSE;
paperMachineHmiCommands.dryingSectionGroup1SteamPressureManualSetpoint := 0.0;

paperMachineHmiCommands.dryingSectionGroup2SteamPressureAutoMan := FALSE;
paperMachineHmiCommands.dryingSectionGroup2SteamPressureManualSetpoint := 0.0;

paperMachineHmiCommands.dryingSectionGroup3SteamPressureAutoMan := FALSE;
paperMachineHmiCommands.dryingSectionGroup3SteamPressureManualSetpoint := 0.0;


//Reset first scan flag
firstScan := FALSE;
END_METHOD

METHOD _100_FormingBoardControl
VAR_INPUT
END_VAR
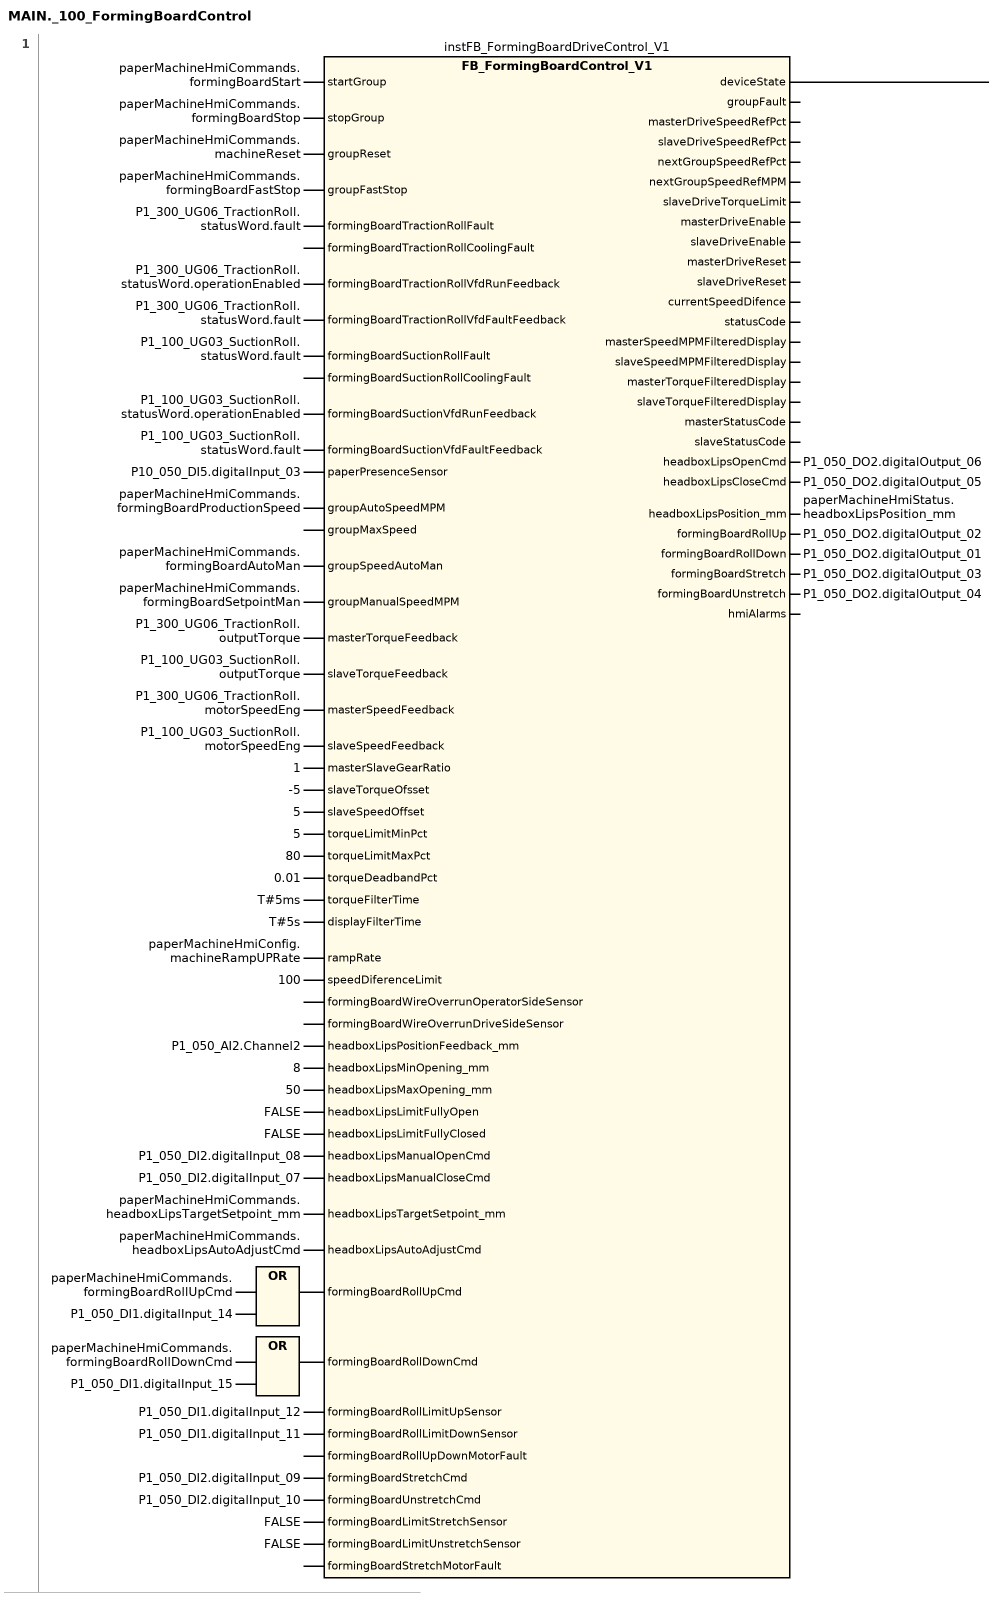
// NETWORK 1
instFB_FormingBoardDriveControl_V1(
    startGroup := paperMachineHmiCommands.formingBoardStart,
    stopGroup := paperMachineHmiCommands.formingBoardStop,
    groupReset := paperMachineHmiCommands.machineReset,
    groupFastStop := paperMachineHmiCommands.formingBoardFastStop,
    formingBoardTractionRollFault := P1_300_UG06_TractionRoll.statusWord.fault,
    formingBoardTractionRollVfdRunFeedback := P1_300_UG06_TractionRoll.statusWord.operationEnabled,
    formingBoardTractionRollVfdFaultFeedback := P1_300_UG06_TractionRoll.statusWord.fault,
    formingBoardSuctionRollFault := P1_100_UG03_SuctionRoll.statusWord.fault,
    formingBoardSuctionVfdRunFeedback := P1_100_UG03_SuctionRoll.statusWord.operationEnabled,
    formingBoardSuctionVfdFaultFeedback := P1_100_UG03_SuctionRoll.statusWord.fault,
    paperPresenceSensor := P10_050_DI5.digitalInput_03,
    groupAutoSpeedMPM := paperMachineHmiCommands.formingBoardProductionSpeed,
    groupSpeedAutoMan := paperMachineHmiCommands.formingBoardAutoMan,
    groupManualSpeedMPM := paperMachineHmiCommands.formingBoardSetpointMan,
    masterTorqueFeedback := P1_300_UG06_TractionRoll.outputTorque,
    slaveTorqueFeedback := P1_100_UG03_SuctionRoll.outputTorque,
    masterSpeedFeedback := P1_300_UG06_TractionRoll.motorSpeedEng,
    slaveSpeedFeedback := P1_100_UG03_SuctionRoll.motorSpeedEng,
    masterSlaveGearRatio := 1,
    slaveTorqueOfsset := -5,
    slaveSpeedOffset := 5,
    torqueLimitMinPct := 5,
    torqueLimitMaxPct := 80,
    torqueDeadbandPct := 0.01,
    torqueFilterTime := T#5ms,
    displayFilterTime := T#5s,
    rampRate := paperMachineHmiConfig.machineRampUPRate,
    speedDiferenceLimit := 100,
    headboxLipsPositionFeedback_mm := P1_050_AI2.Channel2,
    headboxLipsMinOpening_mm := 8,
    headboxLipsMaxOpening_mm := 50,
    headboxLipsLimitFullyOpen := FALSE,
    headboxLipsLimitFullyClosed := FALSE,
    headboxLipsManualOpenCmd := P1_050_DI2.digitalInput_08,
    headboxLipsManualCloseCmd := P1_050_DI2.digitalInput_07,
    headboxLipsTargetSetpoint_mm := paperMachineHmiCommands.headboxLipsTargetSetpoint_mm,
    headboxLipsAutoAdjustCmd := paperMachineHmiCommands.headboxLipsAutoAdjustCmd,
    formingBoardRollUpCmd := paperMachineHmiCommands.formingBoardRollUpCmd OR P1_050_DI1.digitalInput_14,
    formingBoardRollDownCmd := paperMachineHmiCommands.formingBoardRollDownCmd OR P1_050_DI1.digitalInput_15,
    formingBoardRollLimitUpSensor := P1_050_DI1.digitalInput_12,
    formingBoardRollLimitDownSensor := P1_050_DI1.digitalInput_11,
    formingBoardStretchCmd := P1_050_DI2.digitalInput_09,
    formingBoardUnstretchCmd := P1_050_DI2.digitalInput_10,
    formingBoardLimitStretchSensor := FALSE,
    formingBoardLimitUnstretchSensor := FALSE,
    headboxLipsOpenCmd => P1_050_DO2.digitalOutput_06,
    headboxLipsCloseCmd => P1_050_DO2.digitalOutput_05,
    headboxLipsPosition_mm => paperMachineHmiStatus.headboxLipsPosition_mm,
    formingBoardRollUp => P1_050_DO2.digitalOutput_02,
    formingBoardRollDown => P1_050_DO2.digitalOutput_01,
    formingBoardStretch => P1_050_DO2.digitalOutput_03,
    formingBoardUnstretch => P1_050_DO2.digitalOutput_04); // FB_FormingBoardControl_V1

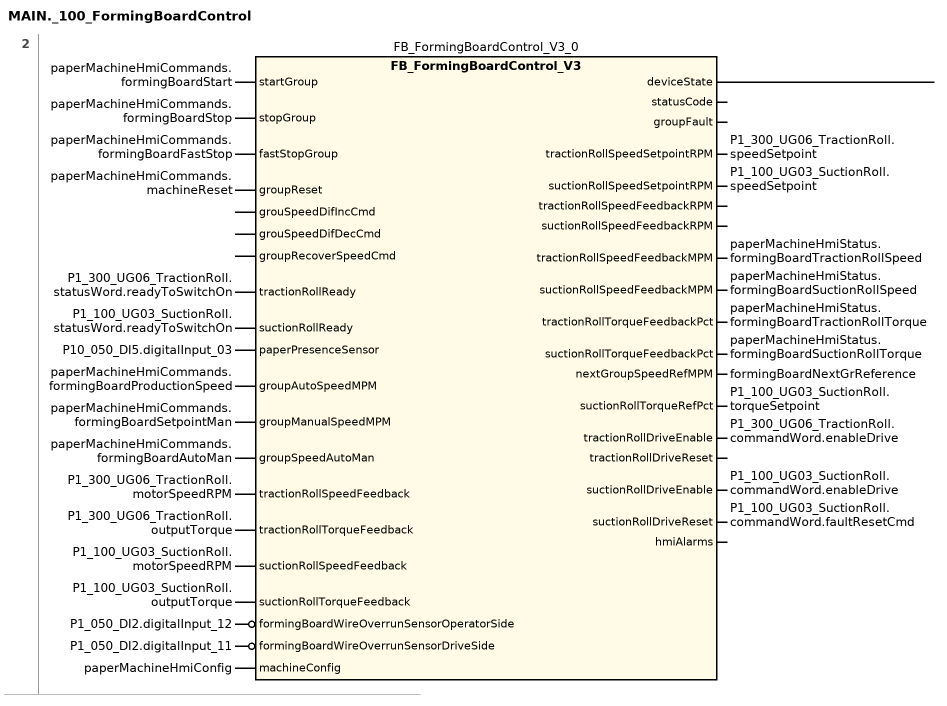
// NETWORK 2
FB_FormingBoardControl_V3_0(
    startGroup := paperMachineHmiCommands.formingBoardStart,
    stopGroup := paperMachineHmiCommands.formingBoardStop,
    fastStopGroup := paperMachineHmiCommands.formingBoardFastStop,
    groupReset := paperMachineHmiCommands.machineReset,
    tractionRollReady := P1_300_UG06_TractionRoll.statusWord.readyToSwitchOn,
    suctionRollReady := P1_100_UG03_SuctionRoll.statusWord.readyToSwitchOn,
    paperPresenceSensor := P10_050_DI5.digitalInput_03,
    groupAutoSpeedMPM := paperMachineHmiCommands.formingBoardProductionSpeed,
    groupManualSpeedMPM := paperMachineHmiCommands.formingBoardSetpointMan,
    groupSpeedAutoMan := paperMachineHmiCommands.formingBoardAutoMan,
    tractionRollSpeedFeedback := P1_300_UG06_TractionRoll.motorSpeedRPM,
    tractionRollTorqueFeedback := P1_300_UG06_TractionRoll.outputTorque,
    suctionRollSpeedFeedback := P1_100_UG03_SuctionRoll.motorSpeedRPM,
    suctionRollTorqueFeedback := P1_100_UG03_SuctionRoll.outputTorque,
    formingBoardWireOverrunSensorOperatorSide := NOT P1_050_DI2.digitalInput_12,
    formingBoardWireOverrunSensorDriveSide := NOT P1_050_DI2.digitalInput_11,
    machineConfig := paperMachineHmiConfig,
    tractionRollSpeedSetpointRPM => P1_300_UG06_TractionRoll.speedSetpoint,
    suctionRollSpeedSetpointRPM => P1_100_UG03_SuctionRoll.speedSetpoint,
    tractionRollSpeedFeedbackMPM => paperMachineHmiStatus.formingBoardTractionRollSpeed,
    suctionRollSpeedFeedbackMPM => paperMachineHmiStatus.formingBoardSuctionRollSpeed,
    tractionRollTorqueFeedbackPct => paperMachineHmiStatus.formingBoardTractionRollTorque,
    suctionRollTorqueFeedbackPct => paperMachineHmiStatus.formingBoardSuctionRollTorque,
    nextGroupSpeedRefMPM => formingBoardNextGrReference,
    suctionRollTorqueRefPct => P1_100_UG03_SuctionRoll.torqueSetpoint,
    tractionRollDriveEnable => P1_300_UG06_TractionRoll.commandWord.enableDrive,
    suctionRollDriveEnable => P1_100_UG03_SuctionRoll.commandWord.enableDrive,
    suctionRollDriveReset => P1_100_UG03_SuctionRoll.commandWord.faultResetCmd); // FB_FormingBoardControl_V3
END_METHOD

METHOD _110_FormingBoardAux
VAR_INPUT
END_VAR
(*


	formingTailCutterNozzleStartCmd   : BOOL; 
	formingTailCutterNozzleStopCmd   : BOOL; 
	formingWireShowerStartCmd : BOOL; 
	formingWireShowerStopCmd : BOOL; 	

*)
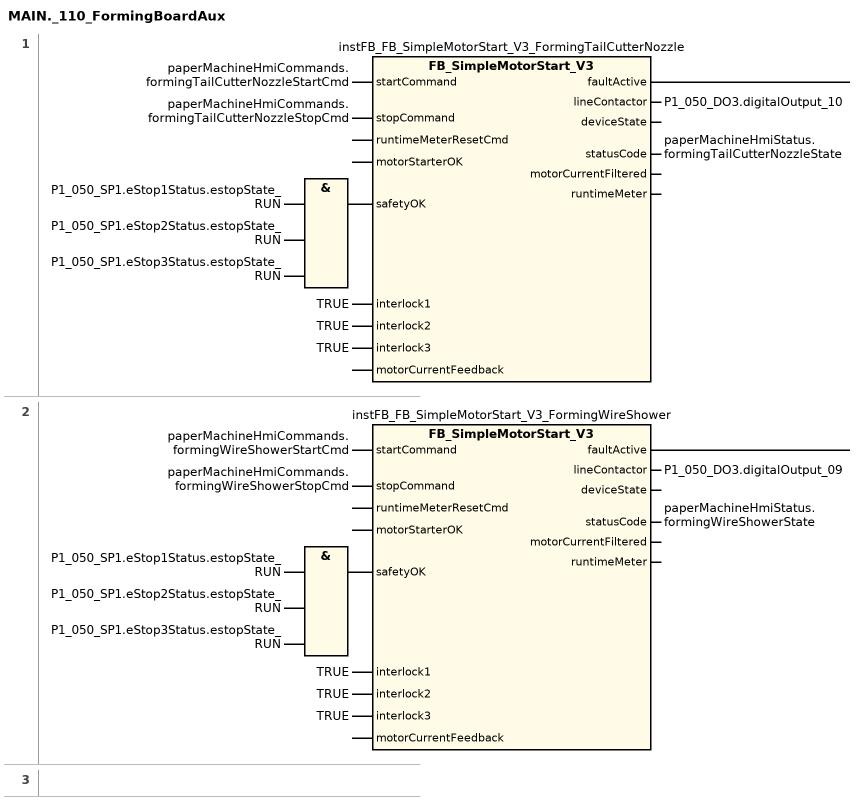
// NETWORK 1
instFB_FB_SimpleMotorStart_V3_FormingTailCutterNozzle(
    startCommand := paperMachineHmiCommands.formingTailCutterNozzleStartCmd,
    stopCommand := paperMachineHmiCommands.formingTailCutterNozzleStopCmd,
    safetyOK := P1_050_SP1.eStop1Status.estopState_RUN AND P1_050_SP1.eStop2Status.estopState_RUN AND P1_050_SP1.eStop3Status.estopState_RUN,
    interlock1 := TRUE,
    interlock2 := TRUE,
    interlock3 := TRUE,
    lineContactor => P1_050_DO3.digitalOutput_10,
    statusCode => paperMachineHmiStatus.formingTailCutterNozzleState); // FB_SimpleMotorStart_V3

// NETWORK 2
instFB_FB_SimpleMotorStart_V3_FormingWireShower(
    startCommand := paperMachineHmiCommands.formingWireShowerStartCmd,
    stopCommand := paperMachineHmiCommands.formingWireShowerStopCmd,
    safetyOK := P1_050_SP1.eStop1Status.estopState_RUN AND P1_050_SP1.eStop2Status.estopState_RUN AND P1_050_SP1.eStop3Status.estopState_RUN,
    interlock1 := TRUE,
    interlock2 := TRUE,
    interlock3 := TRUE,
    lineContactor => P1_050_DO3.digitalOutput_09,
    statusCode => paperMachineHmiStatus.formingWireShowerState); // FB_SimpleMotorStart_V3

// NETWORK 3
END_METHOD

METHOD _200_PressSectionControl
VAR_INPUT
END_VAR
(*

P1_200_UG01();	//First press group master motor
P1_200_UG02();	//First press group slave motor
	
P1_300_UG01();	//First drying group master motor
P1_300_UG02();	//First drying group slave 1
P1_300_UG03();	//First drying group slave 2
	
P1_400_UG01();	//Second drying group master motor
P1_400_UG02();	//Second drying group slave 1
P1_400_UG03();	//Second drying group slave 2

*)
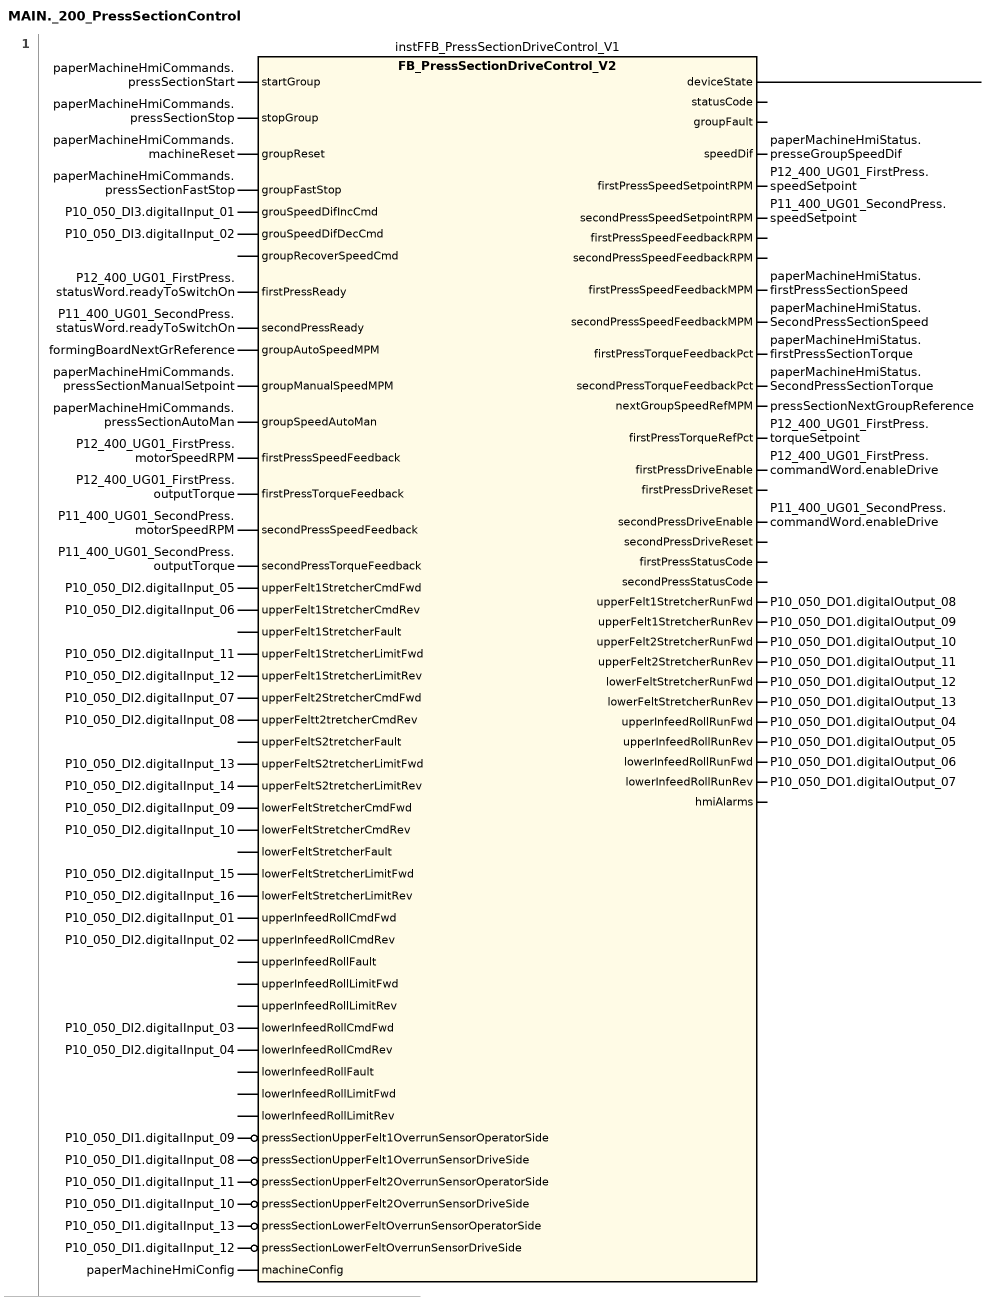
// NETWORK 1
instFFB_PressSectionDriveControl_V1(
    startGroup := paperMachineHmiCommands.pressSectionStart,
    stopGroup := paperMachineHmiCommands.pressSectionStop,
    groupReset := paperMachineHmiCommands.machineReset,
    groupFastStop := paperMachineHmiCommands.pressSectionFastStop,
    grouSpeedDifIncCmd := P10_050_DI3.digitalInput_01,
    grouSpeedDifDecCmd := P10_050_DI3.digitalInput_02,
    firstPressReady := P12_400_UG01_FirstPress.statusWord.readyToSwitchOn,
    secondPressReady := P11_400_UG01_SecondPress.statusWord.readyToSwitchOn,
    groupAutoSpeedMPM := formingBoardNextGrReference,
    groupManualSpeedMPM := paperMachineHmiCommands.pressSectionManualSetpoint,
    groupSpeedAutoMan := paperMachineHmiCommands.pressSectionAutoMan,
    firstPressSpeedFeedback := P12_400_UG01_FirstPress.motorSpeedRPM,
    firstPressTorqueFeedback := P12_400_UG01_FirstPress.outputTorque,
    secondPressSpeedFeedback := P11_400_UG01_SecondPress.motorSpeedRPM,
    secondPressTorqueFeedback := P11_400_UG01_SecondPress.outputTorque,
    upperFelt1StretcherCmdFwd := P10_050_DI2.digitalInput_05,
    upperFelt1StretcherCmdRev := P10_050_DI2.digitalInput_06,
    upperFelt1StretcherLimitFwd := P10_050_DI2.digitalInput_11,
    upperFelt1StretcherLimitRev := P10_050_DI2.digitalInput_12,
    upperFelt2StretcherCmdFwd := P10_050_DI2.digitalInput_07,
    upperFeltt2tretcherCmdRev := P10_050_DI2.digitalInput_08,
    upperFeltS2tretcherLimitFwd := P10_050_DI2.digitalInput_13,
    upperFeltS2tretcherLimitRev := P10_050_DI2.digitalInput_14,
    lowerFeltStretcherCmdFwd := P10_050_DI2.digitalInput_09,
    lowerFeltStretcherCmdRev := P10_050_DI2.digitalInput_10,
    lowerFeltStretcherLimitFwd := P10_050_DI2.digitalInput_15,
    lowerFeltStretcherLimitRev := P10_050_DI2.digitalInput_16,
    upperInfeedRollCmdFwd := P10_050_DI2.digitalInput_01,
    upperInfeedRollCmdRev := P10_050_DI2.digitalInput_02,
    lowerInfeedRollCmdFwd := P10_050_DI2.digitalInput_03,
    lowerInfeedRollCmdRev := P10_050_DI2.digitalInput_04,
    pressSectionUpperFelt1OverrunSensorOperatorSide := NOT P10_050_DI1.digitalInput_09,
    pressSectionUpperFelt1OverrunSensorDriveSide := NOT P10_050_DI1.digitalInput_08,
    pressSectionUpperFelt2OverrunSensorOperatorSide := NOT P10_050_DI1.digitalInput_11,
    pressSectionUpperFelt2OverrunSensorDriveSide := NOT P10_050_DI1.digitalInput_10,
    pressSectionLowerFeltOverrunSensorOperatorSide := NOT P10_050_DI1.digitalInput_13,
    pressSectionLowerFeltOverrunSensorDriveSide := NOT P10_050_DI1.digitalInput_12,
    machineConfig := paperMachineHmiConfig,
    speedDif => paperMachineHmiStatus.presseGroupSpeedDif,
    firstPressSpeedSetpointRPM => P12_400_UG01_FirstPress.speedSetpoint,
    secondPressSpeedSetpointRPM => P11_400_UG01_SecondPress.speedSetpoint,
    firstPressSpeedFeedbackMPM => paperMachineHmiStatus.firstPressSectionSpeed,
    secondPressSpeedFeedbackMPM => paperMachineHmiStatus.SecondPressSectionSpeed,
    firstPressTorqueFeedbackPct => paperMachineHmiStatus.firstPressSectionTorque,
    secondPressTorqueFeedbackPct => paperMachineHmiStatus.SecondPressSectionTorque,
    nextGroupSpeedRefMPM => pressSectionNextGroupReference,
    firstPressTorqueRefPct => P12_400_UG01_FirstPress.torqueSetpoint,
    firstPressDriveEnable => P12_400_UG01_FirstPress.commandWord.enableDrive,
    secondPressDriveEnable => P11_400_UG01_SecondPress.commandWord.enableDrive,
    upperFelt1StretcherRunFwd => P10_050_DO1.digitalOutput_08,
    upperFelt1StretcherRunRev => P10_050_DO1.digitalOutput_09,
    upperFelt2StretcherRunFwd => P10_050_DO1.digitalOutput_10,
    upperFelt2StretcherRunRev => P10_050_DO1.digitalOutput_11,
    lowerFeltStretcherRunFwd => P10_050_DO1.digitalOutput_12,
    lowerFeltStretcherRunRev => P10_050_DO1.digitalOutput_13,
    upperInfeedRollRunFwd => P10_050_DO1.digitalOutput_04,
    upperInfeedRollRunRev => P10_050_DO1.digitalOutput_05,
    lowerInfeedRollRunFwd => P10_050_DO1.digitalOutput_06,
    lowerInfeedRollRunRev => P10_050_DO1.digitalOutput_07); // FB_PressSectionDriveControl_V2
END_METHOD

METHOD _500_DryingSectionGroup1DriveControl
VAR_INPUT
END_VAR

(*

	dryingSectionGroup1SteamPressureAutoMan : BOOL;  // Recovery speed increment [m/min or %] (Incremento de recuperação Grupo 1)
	dryingSectionGroup1SteamPressureAutoSetpoint : REAL;  // Recovery speed increment [m/min or %] (Incremento de recuperação Grupo 1)
	dryingSectionGroup1SteamPressureManualSetpoint : REAL;  // Recovery speed increment [m/min or %] (Incremento de recuperação Grupo 1)
	
